            (* RETRY DISABLED - No retry count limit checking
            // Check if try count exceeds limit after incrementing
            // RetryCount specifies maximum number of attempts allowed
            // RetryCount=0 means 1 attempt, RetryCount=1 means 1 attempt, RetryCount=2 means 2 attempts, etc.
            IF (CommandStatus.CommandTryCount > _ResolveCommandConfiguration().RetryCount) AND
               (_ResolveCommandConfiguration().RetryCount > 0) THEN
                CommandStatus.Result := E_CommandResult.TooManyRequests; // 429
                // Log the TooManyRequests error with command details
                TraceWithSeverity(
                    Message := Tc2_Standard.CONCAT('Command exceeded retry limit: ',
                        Tc2_Standard.CONCAT(CommandStatus.LastCommandMessage,
                        Tc2_Standard.CONCAT(' | TryCount: ',
                        Tc2_Standard.CONCAT(DINT_TO_STRING(CommandStatus.CommandTryCount),
                        Tc2_Standard.CONCAT(' | RetryLimit: ',
                        DINT_TO_STRING(_ResolveCommandConfiguration().RetryCount)))))),
                    Severity := Global.TcEventSeverity.Warning);
                IF __ISVALIDREF(CommandStatus.BaseStatus) THEN
                    CommandStatus.BaseStatus.Error := TRUE;
                                        CommandStatus.BaseStatus.Done := TRUE;  // Complete state always sets Done=TRUE (terminal state)
                                    ELSE
                    TraceWithSeverity(Message := 'Command Base Reference Data Structure not present - see _InitializeReferences', Severity := Global.TcEventSeverity.Error);
                END_IF
                CommandStatus.StepState := E_CommandState.Complete;
                                //iTimer.ResetTimer();
            ELSIF (CommandStatus.CommandTryCount > 1) AND
                  (_ResolveCommandConfiguration().RetryCount = 0) THEN
                // Special case: RetryCount=0 means only 1 attempt allowed
                CommandStatus.Result := E_CommandResult.TooManyRequests; // 429
                // Log the TooManyRequests error for no-retry configuration
                TraceWithSeverity(
                    Message := Tc2_Standard.CONCAT('Command exceeded limit (no retries allowed): ',
                        Tc2_Standard.CONCAT(CommandStatus.LastCommandMessage,
                        Tc2_Standard.CONCAT(' | TryCount: ',
                        DINT_TO_STRING(CommandStatus.CommandTryCount)))),
                    Severity := Global.TcEventSeverity.Warning);
                IF __ISVALIDREF(CommandStatus.BaseStatus) THEN
                    CommandStatus.BaseStatus.Error := TRUE;
                                        CommandStatus.BaseStatus.Done := TRUE;  // Complete state always sets Done=TRUE (terminal state)
                                    ELSE
                    TraceWithSeverity(Message := 'Command Base Reference Data Structure not present - see _InitializeReferences', Severity := Global.TcEventSeverity.Error);
                END_IF
                CommandStatus.StepState := E_CommandState.Complete;
                                //iTimer.ResetTimer();
            END_IF
            *)
        END_IF

    E_CommandState.Execute:
        // Execute state: immediately transition to Monitor (tests expect this progression)
        CommandStatus.StepState := E_CommandState.Monitor;
        
    E_CommandState.Monitor:
        // All commands now monitor for completion condition
        // Check for timeout first (error condition takes priority)
        IF (_iCommandConfiguration <> 0) THEN
            IF CommandStatus.LastCommandElapsedTime >= TIME_TO_LTIME(_iCommandConfiguration.P_CommandConfiguration.TimeoutTime) THEN
                IF __ISVALIDREF(_iCommandConfiguration.P_CommandConfiguration.BaseConfiguration) THEN
                    IF _iCommandConfiguration.P_CommandConfiguration.BaseConfiguration.LogTraceConfiguration.What.xLogToEventLogger THEN
                        TraceWithSeverity(Message := 'Command timeout exceeded', Severity := Global.TcEventSeverity.Error);
                    END_IF
                END_IF
                Complete();  // Handle cleanup and clear Busy flag
                CommandStatus.Result := E_CommandResult.RequestTimeout;  // Override with timeout result
                                IF __ISVALIDREF(CommandStatus.BaseStatus) THEN
                    CommandStatus.BaseStatus.Error := TRUE;  // Set error flag for timeout
                                        CommandStatus.BaseStatus.Done := TRUE;  // Complete state always sets Done=TRUE (terminal state)
                                    ELSE
                    TraceWithSeverity(Message := 'Command Base Reference Data Structure not present - see _InitializeReferences', Severity := Global.TcEventSeverity.Error);
                END_IF
                CommandStatus.StepState := E_CommandState.Complete;  // Transition to Complete state
                            // Check if completion condition is met using resolved configuration (supports fallback)
            ELSIF __ISVALIDREF(_ResolveCommandConfiguration().CompletionCondition) AND_THEN
                  _ResolveCommandConfiguration().CompletionCondition THEN
                // Completion condition met - call Complete() to handle cleanup and transition
                IF NOT SUPER^.BaseStatus.LogTraceStatus.CompletionConditionMetShown THEN
                    TraceWithSeverity(Message := 'Completion condition met', Severity := Global.TcEventSeverity.Info);
                    SUPER^.BaseStatus.LogTraceStatus.CompletionConditionMetShown := TRUE;
                END_IF
                Complete();
                // Set Done flag and Ok result for successful completion (since Complete state won't be processed in this cycle due to REPEAT..UNTIL)
                IF CommandStatus.Result = E_CommandResult.Accepted THEN
                    CommandStatus.Result := E_CommandResult.Ok;
                    IF __ISVALIDREF(CommandStatus.BaseStatus) THEN
                        CommandStatus.BaseStatus.Done := TRUE;
                    ELSE
                        TraceWithSeverity(Message := 'Command Base Reference Data Structure not present - see _InitializeReferences', Severity := Global.TcEventSeverity.Error);
                    END_IF
                END_IF
                CommandStatus.StepState := E_CommandState.Complete;
                            END_IF
        ELSE
            // WARNING: _iCommandConfiguration is null - timeout monitoring disabled, relying on completion condition only
            TraceWithSeverity(Message := 'WARNING: _iCommandConfiguration is null in Monitor state - timeout monitoring disabled', Severity := Global.TcEventSeverity.Warning);
            IF __ISVALIDREF(_ResolveCommandConfiguration().CompletionCondition) AND_THEN
               _ResolveCommandConfiguration().CompletionCondition THEN
			   IF NOT SUPER^.BaseStatus.LogTraceStatus.CompletionConditionMetShown THEN
			       TraceWithSeverity(Message := 'Completion condition met', Severity := Global.TcEventSeverity.Info);
			       SUPER^.BaseStatus.LogTraceStatus.CompletionConditionMetShown := TRUE;
			   END_IF
                // No command configuration but completion condition met
                Complete();
                // Set Done flag and Ok result for successful completion (since Complete state won't be processed in this cycle due to REPEAT..UNTIL)
                IF CommandStatus.Result = E_CommandResult.Accepted THEN
                    CommandStatus.Result := E_CommandResult.Ok;
                    IF __ISVALIDREF(CommandStatus.BaseStatus) THEN
                        CommandStatus.BaseStatus.Done := TRUE;
                    ELSE
                        TraceWithSeverity(Message := 'Command Base Reference Data Structure not present - see _InitializeReferences', Severity := Global.TcEventSeverity.Error);
                    END_IF
                END_IF
                CommandStatus.StepState := E_CommandState.Complete;
                            END_IF
        END_IF
        // Otherwise stay in Monitor state until:
        // 1. CompletionCondition becomes TRUE
        // 2. Component calls Complete() method directly
        // 3. Timeout occurs (checked above)

    E_CommandState.Complete:
        // Stop the timer when entering Complete state
        IF iTimer <> 0 THEN
            iTimer.StopTimer();
        END_IF

        // Only set Ok on successful completion (if no error was already set)
        IF CommandStatus.Result = E_CommandResult.Accepted THEN
            CommandStatus.Result := E_CommandResult.Ok;
                        IF __ISVALIDREF(CommandStatus.BaseStatus) THEN
                CommandStatus.BaseStatus.Done := TRUE;
                            ELSE
                TraceWithSeverity(Message := 'Command Base Reference Data Structure not present - see _InitializeReferences', Severity := Global.TcEventSeverity.Error);
            END_IF
        END_IF
        // Otherwise preserve the existing error result (RequestTimeout, Aborted, etc.)
        // Error results already have Done=TRUE set by the method that created the error


END_CASE
UNTIL (CommandStatus.StepState = E_CommandState.Monitor) OR
      (CommandStatus.StepState = E_CommandState.Complete) OR
      (CommandStatus.StepState = E_CommandState.Idle)
END_REPEAT
END_METHOD

METHOD PRIVATE _ResetCommand
// Policy G: Always clear to complete reset state
IF __ISVALIDREF(CommandStatus.BaseStatus) THEN
	// Verbose logging: Log reset with context before clearing state
	TraceWithSeverity(
		Message := CONCAT(
			CONCAT('Resetting command from StepState: ', _FormatStepStateString(CommandStatus.StepState)),
			CONCAT(' | Result: ', CONCAT(_FormatResultString(CommandStatus.Result),
			CONCAT(' | TryCount: ', DINT_TO_STRING(CommandStatus.CommandTryCount))))
		),
		Severity := Global.TcEventSeverity.Verbose
	);

	CommandStatus.CommandTryCount	:= 0;
	CommandStatus.BaseStatus.Busy	:= FALSE;
	CommandStatus.Result 			:= E_CommandResult.None;
	CommandStatus.BaseStatus.Done	:= FALSE;
	CommandStatus.BaseStatus.Error	:= FALSE;
	CommandStatus.BaseStatus.ErrorID := 0; // Clear error ID per policy G
	CommandStatus.StepState			:= E_CommandState.Idle;
	CommandStatus.PreviousStepState := E_CommandState.Idle; // Reset previous state tracking

	// Reset Complete state cycle counter
	CompleteStateCycles := 0;

	// Reset the command timer to clear elapsed time
	IF iTimer <> 0 THEN
		iTimer.ResetTimer();
	ELSE
		// Timer interface not available - log critical error
		TraceWithSeverity(Message := 'CRITICAL: Timer interface not available during _ResetCommand - elapsed time may not reset!', Severity := Global.TcEventSeverity.Error);
	END_IF

	// Force reset elapsed time tracking to prevent instant timeout on next execution
	// This is a backup in case iTimer is null and ResetTimer() couldn't clear these
	CommandStatus.LastCommandElapsedTime := LTIME#0s;
	CommandStatus.LastCommandTriggerTime := 0;

	// Reset cyclic log spam flags to allow messages on next execution
	CommandStatus.BaseStatus.LogTraceStatus.CmdValidatedShown := FALSE;
	CommandStatus.BaseStatus.LogTraceStatus.CmdValidationFailedShown := FALSE;
	CommandStatus.BaseStatus.LogTraceStatus.CompletionConditionMetShown := FALSE;
	CommandStatus.BaseStatus.LogTraceStatus.InterlockLossShown := FALSE;
	CommandStatus.BaseStatus.LogTraceStatus.ConfigInvalidRefShown := FALSE;
ELSE
	TraceWithSeverity(Message := 'Command Base Reference Data Structure not present - see _InitializeReferences', Severity := Global.TcEventSeverity.Error);
END_IF
END_METHOD

METHOD PROTECTED _ResolveCommandConfiguration : REFERENCE TO ST_CommandConfiguration
VAR
    logEnabled : BOOL;
END_VAR
// Precompute whether we should emit logs
logEnabled := (SUPER^.BaseConfiguration.LogTraceConfiguration.When = E_LogTraceWhen.xRunCyclic)
              AND_THEN SUPER^.BaseConfiguration.LogTraceConfiguration.What.xLogToEventLogger;

// 1) Missing command interface?
IF _iCommandConfiguration = 0 THEN
    IF SUPER^.BaseConfiguration.LogTraceConfiguration.What.xLogToEventLogger AND NOT SUPER^.BaseStatus.LogTraceStatus.ConfigInvalidRefShown THEN
        TraceWithSeverity('Missing I_CommandConfiguration interface', Severity := Global.TcEventSeverity.Error);
        SUPER^.BaseStatus.LogTraceStatus.ConfigInvalidRefShown := TRUE;
    END_IF

// 2) Missing perm-intlk interface?
ELSIF _iPermIntlkConfiguration = 0 THEN
    IF SUPER^.BaseConfiguration.LogTraceConfiguration.What.xLogToEventLogger AND NOT SUPER^.BaseStatus.LogTraceStatus.ConfigInvalidRefShown THEN
        TraceWithSeverity('Missing I_PermIntlkConfiguration interface', Severity := Global.TcEventSeverity.Error);
        SUPER^.BaseStatus.LogTraceStatus.ConfigInvalidRefShown := TRUE;
    END_IF

ELSE
    // Both interfaces non-zero → validate each link in the chain

    // a) Command POU config must exist
    IF NOT __ISVALIDREF(_iCommandConfiguration.P_CommandConfiguration) THEN
        IF SUPER^.BaseConfiguration.LogTraceConfiguration.What.xLogToEventLogger AND NOT SUPER^.BaseStatus.LogTraceStatus.ConfigInvalidRefShown THEN
            TraceWithSeverity('_iCommandConfiguration.P_CommandConfiguration is invalid', Severity := Global.TcEventSeverity.Error);
            SUPER^.BaseStatus.LogTraceStatus.ConfigInvalidRefShown := TRUE;
        END_IF

    // b) PermIntlk POU config must exist
    ELSIF NOT __ISVALIDREF(_iPermIntlkConfiguration.P_PermIntlkConfiguration) THEN
        IF __ISVALIDREF(_iCommandConfiguration.P_CommandConfiguration.BaseConfiguration) THEN
            IF _iCommandConfiguration.P_CommandConfiguration.BaseConfiguration.LogTraceConfiguration.What.xLogToEventLogger AND NOT SUPER^.BaseStatus.LogTraceStatus.ConfigInvalidRefShown THEN
                TraceWithSeverity('_iPermIntlkConfiguration.P_PermIntlkConfiguration is invalid', Severity := Global.TcEventSeverity.Error);
                SUPER^.BaseStatus.LogTraceStatus.ConfigInvalidRefShown := TRUE;
            END_IF
        ELSE
            IF SUPER^.BaseConfiguration.LogTraceConfiguration.What.xLogToEventLogger AND NOT SUPER^.BaseStatus.LogTraceStatus.ConfigInvalidRefShown THEN
                TraceWithSeverity('_iPermIntlkConfiguration.P_PermIntlkConfiguration is invalid', Severity := Global.TcEventSeverity.Error);
                SUPER^.BaseStatus.LogTraceStatus.ConfigInvalidRefShown := TRUE;
            END_IF
        END_IF

    // c) Command BaseConfiguration must exist
    ELSIF NOT __ISVALIDREF(_iCommandConfiguration.P_CommandConfiguration.BaseConfiguration) THEN
        IF SUPER^.BaseConfiguration.LogTraceConfiguration.What.xLogToEventLogger AND NOT SUPER^.BaseStatus.LogTraceStatus.ConfigInvalidRefShown THEN
            TraceWithSeverity('_iCommandConfiguration.P_CommandConfiguration.BaseConfiguration is invalid', Severity := Global.TcEventSeverity.Warning);
            SUPER^.BaseStatus.LogTraceStatus.ConfigInvalidRefShown := TRUE;
        END_IF

    // d) PermIntlk BaseConfiguration must exist
    ELSIF NOT __ISVALIDREF(_iPermIntlkConfiguration.P_PermIntlkConfiguration.BaseConfiguration) THEN
        IF __ISVALIDREF(_iCommandConfiguration.P_CommandConfiguration.BaseConfiguration) THEN
            IF _iCommandConfiguration.P_CommandConfiguration.BaseConfiguration.LogTraceConfiguration.What.xLogToEventLogger AND NOT SUPER^.BaseStatus.LogTraceStatus.ConfigInvalidRefShown THEN
                TraceWithSeverity('_iPermIntlkConfiguration.P_PermIntlkConfiguration.BaseConfiguration is invalid', Severity := Global.TcEventSeverity.Error);
                SUPER^.BaseStatus.LogTraceStatus.ConfigInvalidRefShown := TRUE;
            END_IF
        ELSE
            IF SUPER^.BaseConfiguration.LogTraceConfiguration.What.xLogToEventLogger AND NOT SUPER^.BaseStatus.LogTraceStatus.ConfigInvalidRefShown THEN
                TraceWithSeverity('_iPermIntlkConfiguration.P_PermIntlkConfiguration.BaseConfiguration is invalid', Severity := Global.TcEventSeverity.Error);
                SUPER^.BaseStatus.LogTraceStatus.ConfigInvalidRefShown := TRUE;
            END_IF
        END_IF

    // e) Command InstancePath must exist
    ELSIF NOT __ISVALIDREF(_iCommandConfiguration.P_CommandConfiguration.BaseConfiguration.InstancePath) THEN
        IF __ISVALIDREF(_iCommandConfiguration.P_CommandConfiguration.BaseConfiguration) THEN
            IF _iCommandConfiguration.P_CommandConfiguration.BaseConfiguration.LogTraceConfiguration.What.xLogToEventLogger AND NOT SUPER^.BaseStatus.LogTraceStatus.ConfigInvalidRefShown THEN
                TraceWithSeverity('_iCommandConfiguration.P_CommandConfiguration.BaseConfiguration.InstancePath is invalid', Severity := Global.TcEventSeverity.Error);
                SUPER^.BaseStatus.LogTraceStatus.ConfigInvalidRefShown := TRUE;
            END_IF
        ELSE
            IF SUPER^.BaseConfiguration.LogTraceConfiguration.What.xLogToEventLogger AND NOT SUPER^.BaseStatus.LogTraceStatus.ConfigInvalidRefShown THEN
                TraceWithSeverity('_iCommandConfiguration.P_CommandConfiguration.BaseConfiguration.InstancePath is invalid', Severity := Global.TcEventSeverity.Error);
                SUPER^.BaseStatus.LogTraceStatus.ConfigInvalidRefShown := TRUE;
            END_IF
        END_IF

    // f) PermIntlk InstancePath must exist
    ELSIF NOT __ISVALIDREF(_iPermIntlkConfiguration.P_PermIntlkConfiguration.BaseConfiguration.InstancePath) THEN
        IF __ISVALIDREF(_iCommandConfiguration.P_CommandConfiguration.BaseConfiguration) THEN
            IF _iCommandConfiguration.P_CommandConfiguration.BaseConfiguration.LogTraceConfiguration.What.xLogToEventLogger AND NOT SUPER^.BaseStatus.LogTraceStatus.ConfigInvalidRefShown THEN
                TraceWithSeverity('_iPermIntlkConfiguration.P_PermIntlkConfiguration.BaseConfiguration.InstancePath is invalid', Severity := Global.TcEventSeverity.Error);
                SUPER^.BaseStatus.LogTraceStatus.ConfigInvalidRefShown := TRUE;
            END_IF
        ELSE
            IF SUPER^.BaseConfiguration.LogTraceConfiguration.What.xLogToEventLogger AND NOT SUPER^.BaseStatus.LogTraceStatus.ConfigInvalidRefShown THEN
                TraceWithSeverity('_iPermIntlkConfiguration.P_PermIntlkConfiguration.BaseConfiguration.InstancePath is invalid', Severity := Global.TcEventSeverity.Error);
                SUPER^.BaseStatus.LogTraceStatus.ConfigInvalidRefShown := TRUE;
            END_IF
        END_IF

    ELSE
        // All injected refs are valid — wire them up and return
        _iCommandConfiguration.P_CommandConfiguration.PermIntlkConfiguration 
          REF= _iPermIntlkConfiguration.P_PermIntlkConfiguration;
        _ResolveCommandConfiguration
          REF= _iCommandConfiguration.P_CommandConfiguration;
        CommandStatus.CmdConfigurationResolution   := E_ConfigurationResolution.InjectedInterface;
        CommandStatus.PermIntlkConfigResolution   := E_ConfigurationResolution.InjectedInterface;
        RETURN;
    END_IF

END_IF

// Fallback when any check failed
_ResolveCommandConfiguration REF= LocalCommandConfiguration;
CommandStatus.CmdConfigurationResolution   := E_ConfigurationResolution.Local;
CommandStatus.PermIntlkConfigResolution   := E_ConfigurationResolution.Local;
IF SUPER^.BaseConfiguration.LogTraceConfiguration.What.xLogToEventLogger THEN
    TraceWithSeverity('Using fallback CommandConfiguration', Severity := Global.TcEventSeverity.Info);
END_IF
END_METHOD

METHOD PRIVATE _ResolveCommandStatus : REFERENCE TO ST_CommandStatus
IF CommandStatus.CmdConfigurationResolution = E_ConfigurationResolution.InjectedInterface THEN
	IF _iCommandConfiguration <> 0 THEN
		CommandStatus.ConfigRef REF= _iCommandConfiguration.P_CommandConfiguration;
	END_IF
ELSE
	//Fallback
	CommandStatus.ConfigRef REF= LocalCommandConfiguration;
	IF SUPER^.BaseConfiguration.LogTraceConfiguration.When = E_LogTraceWhen.xRunCyclic AND_THEN 
		SUPER^.BaseConfiguration.LogTraceConfiguration.What.xLogToEventLogger THEN
			TraceWithSeverity(Message := 'Using fallback CommandConfiguration', Severity := Global.TcEventSeverity.Info);
	END_IF
END_IF

_ResolveCommandStatus REF= CommandStatus;
END_METHOD

METHOD PRIVATE _ResolvePermIntlkConfiguration : REFERENCE TO ST_PermIntlkConfiguration
VAR
    logEnabled : BOOL;
END_VAR
// 0) Precompute “should we log?”
logEnabled := (SUPER^.BaseConfiguration.LogTraceConfiguration.When = E_LogTraceWhen.xRunCyclic)
              AND_THEN SUPER^.BaseConfiguration.LogTraceConfiguration.What.xLogToEventLogger;

// 1) No injected interface?
IF _iPermIntlkConfiguration = 0 THEN
    IF SUPER^.BaseConfiguration.LogTraceConfiguration.What.xLogToEventLogger THEN
        TraceWithSeverity('Missing I_PermIntlkConfiguration interface', Severity := Global.TcEventSeverity.Error);
    END_IF

ELSE
    // Only now that _iPermIntlkConfiguration<>0 do we inspect its fields:

    // 2) Does the injected P_PermIntlkConfiguration pointer itself exist?
    IF NOT __ISVALIDREF(_iPermIntlkConfiguration.P_PermIntlkConfiguration) THEN
        IF SUPER^.BaseConfiguration.LogTraceConfiguration.What.xLogToEventLogger THEN
            TraceWithSeverity('_iPermIntlkConfiguration.P_PermIntlkConfiguration is invalid', Severity := Global.TcEventSeverity.Info);
        END_IF

    // 3) Is its BaseConfiguration valid?
    ELSIF NOT __ISVALIDREF(_iPermIntlkConfiguration.P_PermIntlkConfiguration.BaseConfiguration) THEN
        IF SUPER^.BaseConfiguration.LogTraceConfiguration.What.xLogToEventLogger THEN
            TraceWithSeverity('_iPermIntlkConfiguration.P_PermIntlkConfiguration.BaseConfiguration is invalid', Severity := Global.TcEventSeverity.Info);
        END_IF

    // 4) Is its BaseConfiguration.InstancePath valid?
    ELSIF NOT __ISVALIDREF(_iPermIntlkConfiguration.P_PermIntlkConfiguration.BaseConfiguration.InstancePath) THEN
        IF SUPER^.BaseConfiguration.LogTraceConfiguration.What.xLogToEventLogger THEN
            TraceWithSeverity('_iPermIntlkConfiguration.P_PermIntlkConfiguration.BaseConfiguration.InstancePath is invalid', Severity := Global.TcEventSeverity.Info);
        END_IF

    ELSE
        // 5) All injected refs are valid → use it and return
        _ResolvePermIntlkConfiguration 
          REF= _iPermIntlkConfiguration.P_PermIntlkConfiguration;
        CommandStatus.PermIntlkConfigResolution := E_ConfigurationResolution.InjectedInterface;
        RETURN;
    END_IF
END_IF

// 6) Fallback: use local config
_ResolvePermIntlkConfiguration REF= LocalPermIntlkConfiguration;
CommandStatus.PermIntlkConfigResolution    := E_ConfigurationResolution.Local;
IF SUPER^.BaseConfiguration.LogTraceConfiguration.What.xLogToEventLogger THEN
    TraceWithSeverity('Using fallback PermIntlkConfiguration', Severity := Global.TcEventSeverity.Info);
END_IF
END_METHOD

METHOD PROTECTED _UpdateComponentStatus
// Update component with last command executed (if component is available)
IF _iComponent <> 0 THEN
	IF CommandStatus.LastCommandResult <> CommandStatus.Result THEN
		CommandStatus.LastCommandResult := CommandStatus.Result;
		_iComponent.P_ComponentStatus.iLastCommand := THIS^;
	END_IF
ELSE
	// Warning: Component interface not available - cannot update component status
	TraceWithSeverity(Message := 'Warning: _iComponent is null in _UpdateComponentStatus - component status not updated', Severity := Global.TcEventSeverity.Warning);
END_IF
END_METHOD

METHOD PROTECTED _UpdateStatusEdgeTracking
// Override base class method to add CommandStatus-specific edge detection
// This method performs edge detection for both BaseStatus (via SUPER^) and CommandStatus
// Call parent class implementation for BaseStatus edge detection
SUPER^._UpdateStatusEdgeTracking();

// Only perform CommandStatus edge detection if verbose tracing is enabled
IF GPL_Base.PERSISTENT_LOG_LEVEL_MIN > Global.TcEventSeverity.Verbose THEN
	RETURN; // Skip edge detection if verbose level is not enabled
END_IF

// StepState edge detection
IF CommandStatus.StepState <> PreviousCommandStatus.StepState THEN
	TraceWithSeverity(
		Message := CONCAT(
			CONCAT('CommandStatus.StepState: ', _FormatStepStateString(PreviousCommandStatus.StepState)),
			CONCAT(' -> ', _FormatStepStateString(CommandStatus.StepState))
		),
		Severity := Global.TcEventSeverity.Verbose
	);
	PreviousCommandStatus.StepState := CommandStatus.StepState;
END_IF

// Result edge detection
IF CommandStatus.Result <> PreviousCommandStatus.Result THEN
	TraceWithSeverity(
		Message := CONCAT(
			CONCAT('CommandStatus.Result: ', _FormatResultString(PreviousCommandStatus.Result)),
			CONCAT(' -> ', _FormatResultString(CommandStatus.Result))
		),
		Severity := Global.TcEventSeverity.Verbose
	);
	PreviousCommandStatus.Result := CommandStatus.Result;
END_IF

// LastCommandTriggerTime edge detection (command start or reset)
IF CommandStatus.LastCommandTriggerTime <> PreviousCommandStatus.LastCommandTriggerTime THEN
	IF CommandStatus.LastCommandTriggerTime = 0 THEN
		// Trigger time reset to 0 - command has been reset
		TraceWithSeverity(
			Message := 'Command Reset - LastCommandTriggerTime cleared',
			Severity := Global.TcEventSeverity.Verbose
		);
	ELSE
		// Trigger time set to actual time - command has started
		TraceWithSeverity(
			Message := CONCAT(
				'Command Started - LastCommandTriggerTime: ',
				F_FileTimeToString(CommandStatus.LastCommandTriggerTime)
			),
			Severity := Global.TcEventSeverity.Verbose
		);
	END_IF
	PreviousCommandStatus.LastCommandTriggerTime := CommandStatus.LastCommandTriggerTime;
END_IF

// LastCommandCompletionTime edge detection (command complete)
IF CommandStatus.LastCommandCompletionTime <> PreviousCommandStatus.LastCommandCompletionTime THEN
	TraceWithSeverity(
		Message := CONCAT(
			CONCAT('Command Completed - LastCommandCompletionTime: ',
			F_FileTimeToString(CommandStatus.LastCommandCompletionTime)),
			CONCAT(' | ElapsedTime: ', LTIME_TO_STRING(CommandStatus.LastCommandElapsedTime))
		),
		Severity := Global.TcEventSeverity.Verbose
	);
	PreviousCommandStatus.LastCommandCompletionTime := CommandStatus.LastCommandCompletionTime;
END_IF
END_METHOD

METHOD PRIVATE _ValidateCommand
VAR
    maxRetries    : DINT;
    isBusy        : BOOL;
    hasPermissive : BOOL := TRUE;
    traceMessage  : STRING;
END_VAR
// Resolve configuration parameters - uses fallback if injected config is invalid
// RETRY DISABLED: maxRetries := _ResolveCommandConfiguration().RetryCount;

// Check component busy state
isBusy := (_iComponent <> 0) AND_THEN _iComponent.Busy;

// Check component enabled state - disabled components cannot execute commands
IF (_iComponent <> 0) AND_THEN NOT _iComponent.P_BaseStatus.Enabled THEN
    CommandStatus.Result := E_CommandResult.Forbidden;    // 403
        IF __ISVALIDREF(CommandStatus.BaseStatus) THEN
        CommandStatus.BaseStatus.Error := TRUE;
            ELSE
        TraceWithSeverity(Message := 'Command Base Reference Data Structure not present - see _InitializeReferences', Severity := Global.TcEventSeverity.Error);
    END_IF
    traceMessage := 'Component disabled - command execution forbidden';
    RETURN;
END_IF

// Check permissives based on configuration availability
// Allow fallback to local configuration when injected config is missing
IF (_iPermIntlkConfiguration <> 0) AND_THEN
   __ISVALIDREF(_iPermIntlkConfiguration.P_PermIntlkConfiguration) AND
   (iPermIntlk <> 0) THEN
    // Injected permissive configuration available
    IF iPermIntlk.Initialized THEN
        // Ensure permissive is current - CyclicLogic now handles evaluation automatically
        iPermIntlk.CyclicLogic();
        hasPermissive := iPermIntlk.P_OK;
        traceMessage := 'Permissive evaluated based on injected configuration';
    ELSE
        // Allow execution if permissive interface provided but not initialized (fail-open for basic tests)
        hasPermissive := TRUE;
        traceMessage := 'Permissive interface present but not initialized - allowing execution';
    END_IF
ELSE
    // No injected permissive config - use fallback (allow execution)
    hasPermissive := TRUE;
    traceMessage := 'Using local fallback configuration – allowing execution';
END_IF

// Now perform validation checks in order of priority
(* RETRY DISABLED - No retry count validation
// Only check retry count if this is actually a retry (command not in Idle state)
IF (CommandStatus.StepState <> E_CommandState.Idle) AND (CommandStatus.CommandTryCount > maxRetries) THEN
    CommandStatus.Result := E_CommandResult.TooManyRequests; // 429
    // Log the validation failure for too many requests
    TraceWithSeverity(
        Message := Tc2_Standard.CONCAT('Command validation failed - retry count exceeded: ',
            Tc2_Standard.CONCAT(CommandStatus.LastCommandMessage,
            Tc2_Standard.CONCAT(' | TryCount: ',
            Tc2_Standard.CONCAT(DINT_TO_STRING(CommandStatus.CommandTryCount),
            Tc2_Standard.CONCAT(' | MaxRetries: ',
            DINT_TO_STRING(maxRetries)))))),
        Severity := Global.TcEventSeverity.Warning);
    IF __ISVALIDREF(CommandStatus.BaseStatus) THEN
        CommandStatus.BaseStatus.Error := TRUE;  // Set error flag for too many requests
            ELSE
        TraceWithSeverity(Message := 'Command Base Reference Data Structure not present - see _InitializeReferences', Severity := Global.TcEventSeverity.Error);
    END_IF
    traceMessage := 'Retry count exceeded';
ELSIF *)
IF (CommandStatus.StepState = E_CommandState.Idle) AND isBusy THEN
    // Only check component busy when starting from Idle (prevents conflicts with other commands)
    // When resuming from Paused/etc, component will be busy with THIS command, which is expected
    CommandStatus.Result := E_CommandResult.BadRequest;        // 400
        IF __ISVALIDREF(CommandStatus.BaseStatus) THEN
        CommandStatus.BaseStatus.Error := TRUE;  // Set error flag for bad request
            ELSE
        TraceWithSeverity(Message := 'Command Base Reference Data Structure not present - see _InitializeReferences', Severity := Global.TcEventSeverity.Error);
    END_IF
    traceMessage := 'Component busy';
ELSIF NOT hasPermissive THEN
    CommandStatus.Result := E_CommandResult.Forbidden;       // 403
    	IF __ISVALIDREF(CommandStatus.BaseStatus) THEN
  		CommandStatus.BaseStatus.Error := TRUE;  // Set error flag for forbidden
  	ELSE
		TraceWithSeverity(Message := 'Command Base Reference Data Structure not present - see _InitializeReferences', Severity := Global.TcEventSeverity.Error);
	END_IF
    IF traceMessage = '' THEN
        traceMessage := 'Permissive not satisfied';
    END_IF
ELSE
    // Policy H: Do NOT increment try count here - only on actual execution start
    CommandStatus.Result := E_CommandResult.Accepted;      // 202
        IF __ISVALIDREF(CommandStatus.BaseStatus) THEN
        CommandStatus.BaseStatus.Error := FALSE;  // Clear error flag for successful validation
            ELSE
        TraceWithSeverity(Message := 'Command Base Reference Data Structure not present - see _InitializeReferences', Severity := Global.TcEventSeverity.Error);
    END_IF
    traceMessage := 'Validation succeeded – ready to process/queue';
END_IF

// Trace logging if enabled
IF _iCommandConfiguration <> 0 THEN
	IF __ISVALIDREF(_iCommandConfiguration.P_CommandConfiguration.BaseConfiguration) THEN
		IF _iCommandConfiguration.P_CommandConfiguration.BaseConfiguration.LogTraceConfiguration.When = E_LogTraceWhen.xRunCyclic AND_THEN
		   _iCommandConfiguration.P_CommandConfiguration.BaseConfiguration.LogTraceConfiguration.What.xLogToEventLogger THEN

			// Only log validation failures once to prevent spam
			IF (CommandStatus.Result <> E_CommandResult.Accepted) THEN
				IF NOT SUPER^.BaseStatus.LogTraceStatus.CmdValidationFailedShown THEN
					TraceWithSeverity(Message :=
						Tc2_Standard.CONCAT(
							STR1 := TO_STRING(CommandStatus.Result),
							STR2 := Tc2_Standard.CONCAT(STR1 := '; ', STR2 := traceMessage)
						), Severity := Global.TcEventSeverity.Info
					);
					SUPER^.BaseStatus.LogTraceStatus.CmdValidationFailedShown := TRUE;
				END_IF
			ELSE
				// Log successful validation normally (less spam concern)
				TraceWithSeverity(Message :=
					Tc2_Standard.CONCAT(
						STR1 := TO_STRING(CommandStatus.Result),
						STR2 := Tc2_Standard.CONCAT(STR1 := '; ', STR2 := traceMessage)
					), Severity := Global.TcEventSeverity.Info
				);
			END_IF
		END_IF
	ELSE
		TraceWithSeverity(Message := 'P_CommandConfiguration.BaseConfiguration reference invalid in _ValidateCommand method', Severity := Global.TcEventSeverity.Error);
		RETURN;
	END_IF
ELSE
	// WARNING: Validation trace logging disabled - configuration interface is null
	TraceWithSeverity(Message := 'WARNING: _iCommandConfiguration is null in _ValidateCommand - validation trace logging disabled', Severity := Global.TcEventSeverity.Warning);
END_IF
END_METHOD

METHOD CyclicLogic
SUPER^.CyclicLogic();

fbPermIntlk.CyclicLogic();

// Only update timer if interface is available
IF iTimer <> 0 THEN
	fbCmdElapsedTime.CyclicLogic();
ELSE
	// Log error once if timer interface is missing during active command
	IF (CommandStatus.StepState <> E_CommandState.Idle) AND (CommandStatus.StepState <> E_CommandState.Complete) THEN
		TraceWithSeverity(Message := 'CRITICAL: Timer interface not present during active command execution!', Severity := Global.TcEventSeverity.Error);
	END_IF
END_IF

// Track state changes for other purposes (CommandTryCount persists across retries, only cleared by Reset)
IF CommandStatus.PreviousStepState <> CommandStatus.StepState THEN
    CommandStatus.PreviousStepState := CommandStatus.StepState;
END_IF

// Execute state machine progression
_ProcessStateTransitions();

// Update component with last command result
_UpdateComponentStatus();

// Handle auto-reset for successful completions
_HandleAutoReset();

// Monitor interlocks and timeouts
_MonitorInterlocks();

// Perform edge detection for status changes at end of cycle (includes BaseStatus and CommandStatus)
_UpdateStatusEdgeTracking();
END_METHOD

PROPERTY P_CommandConfiguration : REFERENCE TO ST_CommandConfiguration
GET
P_CommandConfiguration REF= _ResolveCommandConfiguration();
END_GET
END_PROPERTY

PROPERTY P_PermIntlkConfiguration : REFERENCE TO ST_PermIntlkConfiguration
GET
P_PermIntlkConfiguration REF= _ResolvePermIntlkConfiguration();
END_GET
END_PROPERTY

END_FUNCTION_BLOCK

// PermIntlk/POUs/FB_PermIntlkCommand
{attribute 'no_explicit_call' := 'do not call this POU directly'}
{attribute 'enable_dynamic_creation'}
FUNCTION_BLOCK FB_PermIntlkCommand EXTENDS FB_PermIntlk
VAR
 	_iCommandConfiguration		: I_CommandConfiguration; // External Dependency
END_VAR

METHOD CyclicLogic
SUPER^.CyclicLogic();
END_METHOD

METHOD InjectCommandConfiguration
VAR_INPUT
    iCommandCfg 	: REFERENCE TO I_CommandConfiguration;
END_VAR
IF iCommandCfg = 0 THEN
	//Can't access Trace configuration on Init; use base config
		IF BaseConfiguration.LogTraceConfiguration.What.xLogToEventLogger THEN
			TraceWithSeverity(Message := 'Null Injected interface for Command Configuration!', Severity := Global.TcEventSeverity.Error);
		END_IF
    RETURN;
END_IF

_iCommandConfiguration := iCommandCfg;
END_METHOD

END_FUNCTION_BLOCK

// PermIntlk/POUs/FB_PermIntlk
{attribute 'no_explicit_call' := 'do not call this POU directly'}
{attribute 'enable_dynamic_creation'}
FUNCTION_BLOCK FB_PermIntlk EXTENDS FB_BaseCyclic IMPLEMENTS I_PermIntlk, I_PermIntlkConfiguration
VAR
 	_iPermIntlkConfiguration	: I_PermIntlkConfiguration; // External Dependency
	PermIntlkConfiguration 		: ST_PermIntlkConfiguration; //Local Reference Fallback	
	PermIntlkIndex				: DINT; // FOR loop, etc.
	PermIntlkLogIndex			: DINT; // FOR loop, etc.
	PermIntlkStatus 			: ST_PermIntlkStatus;

	// Guard flag to prevent duplicate evaluation in same scan
	evaluatedThisScan			: BOOL := FALSE;

	// Dummy interface instances for __QUERYINTERFACE type checking
	iQueryInterfaceCheckPermIntlkConfiguration	: I_PermIntlkConfiguration;
END_VAR

METHOD Evaluate : I_PermIntlk
CyclicLogic();

Evaluate := THIS^;
END_METHOD

{attribute 'monitoring' := 'call'}
PROPERTY FINAL P_OK : BOOL
GET
// Ensure fresh evaluation before returning status (avoid duplicate calls in same scan)
IF NOT evaluatedThisScan THEN
    _EvaluateOK();
    evaluatedThisScan := TRUE;
END_IF
P_OK := _ResolvePermIntlkStatus().PermIntlkOK;
END_GET
END_PROPERTY

PROPERTY P_PermIntlkConfiguration : REFERENCE TO ST_PermIntlkConfiguration
GET
P_PermIntlkConfiguration REF= _ResolvePermIntlkConfiguration();
END_GET
END_PROPERTY

(* Basic component initialization logic*)
METHOD PROTECTED _Initialize : BOOL
VAR
	InterimInit : BOOL;
END_VAR
// Initialize children dependencies first
InterimInit := _InitializeChildrenDependencies();
IF NOT InterimInit THEN
	IF PermIntlkConfiguration.BaseConfiguration.LogTraceConfiguration.What.xLogToEventLogger AND NOT PermIntlkStatus.BaseStatus.LogTraceStatus.InitChildrenFailureShown THEN
		TraceWithSeverity(Message := Tc2_Standard.CONCAT('_InitializeChildrenDependencies Failed at ', __POUNAME()), Severity := Global.TcEventSeverity.Error);
		PermIntlkStatus.BaseStatus.LogTraceStatus.InitChildrenFailureShown := TRUE;
	END_IF
	_Initialize := FALSE;
	RETURN;
END_IF

// Set element indices and resolve configurations
_SetElementIndices();
_ResolvePermIntlkConfiguration();
_ResolvePermIntlkStatus();

// Initialize references second
InterimInit := _InitializeReferences();
IF NOT InterimInit THEN
	IF PermIntlkConfiguration.BaseConfiguration.LogTraceConfiguration.What.xLogToEventLogger AND NOT PermIntlkStatus.BaseStatus.LogTraceStatus.InitReferencesFailureShown THEN
		TraceWithSeverity(Message := Tc2_Standard.CONCAT('_InitializeReferences Failed at ', __POUNAME()), Severity := Global.TcEventSeverity.Error);
		PermIntlkStatus.BaseStatus.LogTraceStatus.InitReferencesFailureShown := TRUE;
	END_IF
	_Initialize := FALSE;
	RETURN;
END_IF

// Set dependency configuration last
InterimInit := _SetDependencyConfiguration();
IF NOT InterimInit THEN
	IF PermIntlkConfiguration.BaseConfiguration.LogTraceConfiguration.What.xLogToEventLogger AND NOT PermIntlkStatus.BaseStatus.LogTraceStatus.InitDependencyConfigFailureShown THEN
		TraceWithSeverity(Message := Tc2_Standard.CONCAT('_SetDependencyConfiguration Failed at ', __POUNAME()), Severity := Global.TcEventSeverity.Error);
		PermIntlkStatus.BaseStatus.LogTraceStatus.InitDependencyConfigFailureShown := TRUE;
	END_IF
	_Initialize := FALSE;
	RETURN;
END_IF

// All initialization steps succeeded
_Initialize := TRUE;
END_METHOD

METHOD PROTECTED _InitializeReferences : BOOL
//Order is important!
BaseConfiguration.InstancePath 					REF= InstancePath;

PermIntlkConfiguration.BaseConfiguration		REF= SUPER^.BaseConfiguration;

PermIntlkStatus.BaseStatus						REF= SUPER^.BaseStatus;

// Use resolved configuration for setting up references
IF PermIntlkStatus.PermIntlkConfigResolution = E_ConfigurationResolution.InjectedInterface THEN
	IF _iPermIntlkConfiguration <> 0 THEN
		PermIntlkConfiguration := _iPermIntlkConfiguration.P_PermIntlkConfiguration;
	END_IF
	PermIntlkStatus.ConfigRef	REF= _iPermIntlkConfiguration.P_PermIntlkConfiguration.PermIntlkObj;
	FOR PermIntlkIndex := GC_PermIntlk.INDEX_CONDITION_MIN TO GC_PermIntlk.INDEX_CONDITION_MAX BY 1 DO
		PermIntlkStatus.ConditionStatus[PermIntlkIndex].PermObj	REF= _iPermIntlkConfiguration.P_PermIntlkConfiguration.PermIntlkObj[PermIntlkIndex];
	END_FOR
ELSE
	PermIntlkStatus.ConfigRef	REF= PermIntlkConfiguration.PermIntlkObj;
	FOR PermIntlkIndex := GC_PermIntlk.INDEX_CONDITION_MIN TO GC_PermIntlk.INDEX_CONDITION_MAX BY 1 DO
		PermIntlkConfiguration.PermIntlkObj[PermIntlkIndex].Condition REF= PermIntlkStatus.PermIntlkConditionAlwaysFalse;
		PermIntlkStatus.ConditionStatus[PermIntlkIndex].PermObj	REF= PermIntlkConfiguration.PermIntlkObj[PermIntlkIndex];
	END_FOR
END_IF

_InitializeReferences 							:= TRUE; // apply at end of all reference initialization
END_METHOD

METHOD PROTECTED _SetElementIndices
IF (_iPermIntlkConfiguration <> 0) AND __QUERYINTERFACE(_iPermIntlkConfiguration, iQueryInterfaceCheckPermIntlkConfiguration) THEN
	FOR PermIntlkIndex := GC_PermIntlk.INDEX_CONDITION_MIN TO GC_PermIntlk.INDEX_CONDITION_MAX BY 1 DO
		IF _iPermIntlkConfiguration.P_PermIntlkConfiguration.PermIntlkObj[PermIntlkIndex].Index = 0 THEN
			_iPermIntlkConfiguration.P_PermIntlkConfiguration.PermIntlkObj[PermIntlkIndex].Index := PermIntlkIndex;
		END_IF
	END_FOR
END_IF
END_METHOD

METHOD PRIVATE _EvaluateConfiguration
VAR
	resolvedConfig : REFERENCE TO ST_PermIntlkConfiguration;
	previousResolution : E_ConfigurationResolution;
END_VAR
// Store previous resolution to detect changes
previousResolution := PermIntlkStatus.PermIntlkConfigResolution;

// Get the resolved configuration (injected or local)
resolvedConfig REF= _ResolvePermIntlkConfiguration();

// If configuration resolution changed, update references
IF PermIntlkStatus.PermIntlkConfigResolution <> previousResolution THEN
	_InitializeReferences();
END_IF

FOR PermIntlkLogIndex := GC_PermIntlk.INDEX_CONDITION_MIN TO GC_PermIntlk.INDEX_CONDITION_MAX BY 1 DO

	IF (resolvedConfig.PermIntlkObj[PermIntlkLogIndex].Description <> '') AND
		(resolvedConfig.PermIntlkObj[PermIntlkLogIndex].Description <> 'PermIntlk Condition Not Configured') THEN
		PermIntlkStatus.ConditionStatus[PermIntlkLogIndex].Configured := TRUE;
	END_IF

	//Evaluate Permissive Condition=>Status - references already set up in _InitializeReferences
	_LogMessage(Index := PermIntlkLogIndex);

END_FOR
END_METHOD

METHOD PRIVATE _EvaluateOK
VAR_INST
	PermOKMsgTrig		: Tc2_Standard.R_TRIG;
	PermIntlkLostTrig	: Tc2_Standard.F_TRIG;
END_VAR
VAR
	hasConfiguredConditions : BOOL := FALSE;
	resolvedConfig : REFERENCE TO ST_PermIntlkConfiguration;
END_VAR
// Get the resolved configuration (injected or local)
resolvedConfig REF= _ResolvePermIntlkConfiguration();

// Initialize result based on mode
IF resolvedConfig.Mode = E_ModePermIntlk.IfAnyConditionMet THEN
	PermIntlkStatus.PermIntlkOK := FALSE; // In "Any" mode, assume FALSE until we find a TRUE condition
ELSE
	PermIntlkStatus.PermIntlkOK := TRUE;  // In "All" mode, assume TRUE until we find a FALSE condition
END_IF

FOR PermIntlkIndex := GC_PermIntlk.INDEX_CONDITION_MIN TO GC_PermIntlk.INDEX_CONDITION_MAX BY 1 DO
	
	IF __ISVALIDREF(PermIntlkStatus.ConditionStatus[PermIntlkIndex].PermObj) AND PermIntlkStatus.ConditionStatus[PermIntlkIndex].Configured THEN
		
		IF __ISVALIDREF(PermIntlkStatus.ConditionStatus[PermIntlkIndex].PermObj.Condition) THEN
			hasConfiguredConditions := TRUE;
			IF resolvedConfig.Mode = E_ModePermIntlk.IfAllConditionsMet THEN
				IF NOT PermIntlkStatus.ConditionStatus[PermIntlkIndex].PermObj.Condition THEN
					PermIntlkStatus.PermIntlkOK := FALSE;				
					EXIT;
				END_IF
			ELSIF resolvedConfig.Mode = E_ModePermIntlk.IfAnyConditionMet THEN
				IF PermIntlkStatus.ConditionStatus[PermIntlkIndex].PermObj.Condition THEN
					PermIntlkStatus.PermIntlkOK := TRUE;				
					EXIT;
				END_IF
			END_IF
		ELSE
			PermIntlkStatus.ConditionStatus[PermIntlkIndex].PermObj.Condition REF= PermIntlkStatus.PermIntlkConditionAlwaysFalse;
			TraceWithSeverity(Message := 'Using Injected Interface, but no valid condition reference was supplied - PermIntlk Default Failure', Severity := Global.TcEventSeverity.Error);
		END_IF
	END_IF

END_FOR

// If no configured conditions exist, default to TRUE (safe state)
IF NOT hasConfiguredConditions THEN
	PermIntlkStatus.PermIntlkOK := TRUE;
END_IF

IF SUPER^.BaseConfiguration.LogTraceConfiguration.When = E_LogTraceWhen.xRunCyclic AND_THEN
	SUPER^.BaseConfiguration.LogTraceConfiguration.What.xLogToEventLogger THEN

		PermOKMsgTrig(CLK := PermIntlkStatus.PermIntlkOK);
		PermIntlkLostTrig(CLK := NOT PermIntlkStatus.PermIntlkOK);

		IF PermOKMsgTrig.Q THEN
			SUPER^.TraceWithSeverity(Message := 'Permissive OK ', Severity := Global.TcEventSeverity.Info);
		END_IF

		IF PermIntlkLostTrig.Q THEN
			SUPER^.TraceWithSeverity(Message := 'Interlock Lost ', Severity := Global.TcEventSeverity.Error);
		END_IF

END_IF
END_METHOD

METHOD PROTECTED _LogMessage
VAR_INPUT
	Index : DINT;
END_VAR
//Build output message
IF SUPER^.BaseConfiguration.LogTraceConfiguration.When = E_LogTraceWhen.xRunCyclic AND_THEN
		SUPER^.BaseConfiguration.LogTraceConfiguration.What.xLogToEventLogger THEN
			IF __ISVALIDREF(PermIntlkStatus.ConditionStatus[Index].PermObj) THEN
				// Check if Condition reference is valid before accessing it
				IF __ISVALIDREF(PermIntlkStatus.ConditionStatus[Index].PermObj.Condition) THEN
					IF NOT PermIntlkStatus.ConditionStatus[Index].PermObj.Condition THEN
						IF PermIntlkStatus.ConditionStatus[Index].Configured THEN
							IF NOT PermIntlkStatus.BaseStatus.LogTraceStatus.PermIntlkConditionFailureShown THEN
								PermIntlkStatus.ConditionStatus[Index].ConditionMessage := 'Permissive Condition Missing: ';
								_PermMsgIndexForMessage(Index := Index);
								PermIntlkStatus.ConditionStatus[Index].ConditionMessage := Tc2_Standard.CONCAT(STR1 := PermIntlkStatus.ConditionStatus[Index].ConditionMessage, STR2 := ' ');
								PermIntlkStatus.ConditionStatus[Index].ConditionMessage := Tc2_Standard.CONCAT(STR1 := PermIntlkStatus.ConditionStatus[Index].ConditionMessage, STR2 := PermIntlkStatus.ConditionStatus[Index].PermObj.Description);
								SUPER^.TraceWithSeverity(Message := PermIntlkStatus.ConditionStatus[Index].ConditionMessage, Severity := Global.TcEventSeverity.Error);
								PermIntlkStatus.BaseStatus.LogTraceStatus.PermIntlkConditionFailureShown := TRUE;
							END_IF
						ELSE
							IF NOT PermIntlkStatus.BaseStatus.LogTraceStatus.PermIntlkConditionFailureShown THEN
								PermIntlkStatus.ConditionStatus[Index].ConditionMessage := 'Permissive Description Missing.  Configure permissive: ';
								_PermMsgIndexForMessage(Index := Index);
								SUPER^.TraceWithSeverity(Message := PermIntlkStatus.ConditionStatus[Index].ConditionMessage, Severity := Global.TcEventSeverity.Warning);
								PermIntlkStatus.BaseStatus.LogTraceStatus.PermIntlkConditionFailureShown := TRUE;
							END_IF
						END_IF
					END_IF
				ELSE
					// Condition reference is invalid
					IF PermIntlkStatus.ConditionStatus[Index].Configured THEN
						IF NOT PermIntlkStatus.BaseStatus.LogTraceStatus.PermIntlkConditionFailureShown THEN
							PermIntlkStatus.ConditionStatus[Index].ConditionMessage := 'Permissive Condition Reference Invalid for Index: ';
							_PermMsgIndexForMessage(Index := Index);
							SUPER^.TraceWithSeverity(Message := PermIntlkStatus.ConditionStatus[Index].ConditionMessage, Severity := Global.TcEventSeverity.Error);
							PermIntlkStatus.BaseStatus.LogTraceStatus.PermIntlkConditionFailureShown := TRUE;
						END_IF
					END_IF
				END_IF
			END_IF
// ELSE // logs a message regardless of configuration, due to critical Permissive Data Reference missing
// 	PermIntlkStatus.PermissiveStatusMessage := 'Permissive Missing Reference to Component Log Trace Configuration.  Initialize Component Permissive Data Reference';
// 	SUPER^.Trace(Message := PermIntlkStatus.PermissiveStatusMessage);
END_IF
END_METHOD

METHOD PROTECTED _PermMsgIndexForMessage
VAR_INPUT
	Index : DINT;
END_VAR
PermIntlkStatus.ConditionStatus[Index].ConditionMessage := Tc2_Standard.CONCAT(STR1 := PermIntlkStatus.ConditionStatus[Index].ConditionMessage, STR2 := ' Index:');				
PermIntlkStatus.ConditionStatus[Index].ConditionMessage := Tc2_Standard.CONCAT(STR1 := PermIntlkStatus.ConditionStatus[Index].ConditionMessage, STR2 := UDINT_TO_STRING(PermIntlkStatus.ConditionStatus[Index].PermObj.Index));
END_METHOD

METHOD PROTECTED _ResolvePermIntlkConfiguration : REFERENCE TO ST_PermIntlkConfiguration
VAR
    logEnabled : BOOL;
END_VAR
// Precompute whether we should log
logEnabled := (SUPER^.BaseConfiguration.LogTraceConfiguration.When = E_LogTraceWhen.xRunCyclic)
              AND_THEN SUPER^.BaseConfiguration.LogTraceConfiguration.What.xLogToEventLogger;

// If no interface at all, log and fall through to fallback
IF _iPermIntlkConfiguration = 0 THEN
    IF logEnabled THEN
        TraceWithSeverity('Missing I_PermIntlkConfiguration interface', Severity := Global.TcEventSeverity.Error);
    END_IF

ELSE
    // Only now that _iPermIntlkConfiguration<>0 do we inspect its fields:
    IF NOT __ISVALIDREF(_iPermIntlkConfiguration.P_PermIntlkConfiguration) THEN
        IF logEnabled THEN
            TraceWithSeverity('_iPermIntlkConfiguration.P_PermIntlkConfiguration is invalid', Severity := Global.TcEventSeverity.Info);
        END_IF

    // Optional: BaseConfiguration validation (non-blocking for basic functionality)
    ELSIF NOT __ISVALIDREF(_iPermIntlkConfiguration.P_PermIntlkConfiguration.BaseConfiguration) THEN
        IF logEnabled THEN
            TraceWithSeverity('BaseConfiguration is invalid - using injected interface anyway', Severity := Global.TcEventSeverity.Warning);
        END_IF
        // Continue to use injected interface despite missing BaseConfiguration
        _ResolvePermIntlkConfiguration REF= _iPermIntlkConfiguration.P_PermIntlkConfiguration;
        PermIntlkStatus.PermIntlkConfigResolution := E_ConfigurationResolution.InjectedInterface;
        RETURN;

    ELSIF NOT __ISVALIDREF(_iPermIntlkConfiguration.P_PermIntlkConfiguration.BaseConfiguration.InstancePath) THEN
        IF logEnabled THEN
            TraceWithSeverity('InstancePath is invalid - using injected interface anyway', Severity := Global.TcEventSeverity.Warning);
        END_IF
        // Continue to use injected interface despite missing InstancePath
        _ResolvePermIntlkConfiguration REF= _iPermIntlkConfiguration.P_PermIntlkConfiguration;
        PermIntlkStatus.PermIntlkConfigResolution := E_ConfigurationResolution.InjectedInterface;
        RETURN;

    ELSE
        // All injected refs are valid → return it
        _ResolvePermIntlkConfiguration REF= _iPermIntlkConfiguration.P_PermIntlkConfiguration;
        PermIntlkStatus.PermIntlkConfigResolution := E_ConfigurationResolution.InjectedInterface;
        RETURN;
    END_IF
END_IF

// Fallback path when either interface=0 or any validity check failed:
_ResolvePermIntlkConfiguration REF= PermIntlkConfiguration;
PermIntlkStatus.PermIntlkConfigResolution := E_ConfigurationResolution.Local;
IF logEnabled THEN
    TraceWithSeverity('Using fallback PermIntlkConfiguration', Severity := Global.TcEventSeverity.Info);
END_IF
END_METHOD

METHOD PROTECTED _ResolvePermIntlkStatus : REFERENCE TO ST_PermIntlkStatus
// FOR PermIntlkIndex := LOWER_BOUND(PermIntlkStatus.ConditionStatus,1) TO UPPER_BOUND(PermIntlkStatus.ConditionStatus,1) BY 1 DO
// 	IF __ISVALIDREF(PermIntlkStatus.BaseStatus) AND __ISVALIDREF(PermIntlkStatus.ConfigRef) AND __ISVALIDREF(PermIntlkStatus.ConditionStatus[PermIntlkIndex].PermObj) THEN
// 		_ResolvePermIntlkStatus REF= PermIntlkStatus;		
// 	END_IF
// END_FOR

IF PermIntlkStatus.PermIntlkConfigResolution = E_ConfigurationResolution.InjectedInterface THEN
	PermIntlkStatus.ConfigRef REF= _iPermIntlkConfiguration.P_PermIntlkConfiguration.PermIntlkObj;
ELSE
	PermIntlkStatus.ConfigRef REF= PermIntlkConfiguration.PermIntlkObj;
END_IF

_ResolvePermIntlkStatus REF= PermIntlkStatus;
END_METHOD

METHOD PROTECTED _ConfigurationCyclic
SUPER^._ConfigurationCyclic();

_EvaluateConfiguration();
END_METHOD

METHOD CyclicLogic
SUPER^.CyclicLogic();

// Reset guard flag at start of new scan cycle
evaluatedThisScan := FALSE;

// Always evaluate permissive state on every cycle
_EvaluateOK();
evaluatedThisScan := TRUE;
END_METHOD

METHOD InjectPermIntlkConfiguration
VAR_INPUT
    iPermIntlkCfg 	: I_PermIntlkConfiguration;
END_VAR
// Allow injecting null to clear the interface (for runtime config loss scenarios)
_iPermIntlkConfiguration := iPermIntlkCfg;

IF iPermIntlkCfg = 0 THEN
	//Log warning about null interface - will fall back to local configuration
		TraceWithSeverity(Message := 'Null Injected interface for PermIntlk Configuration - using local fallback', Severity := Global.TcEventSeverity.Warning);
END_IF
END_METHOD

PROPERTY P_PermIntlkStatus : REFERENCE TO ST_PermIntlkStatus
GET
P_PermIntlkStatus REF= PermIntlkStatus;
END_GET
END_PROPERTY

METHOD ReinitObjects
VAR
	 InitPermIntlk 	: ST_PermIntlkConfigurationCondition;
END_VAR
FOR PermIntlkIndex := GC_PermIntlk.INDEX_CONDITION_MIN TO GC_PermIntlk.INDEX_CONDITION_MAX DO
	InitPermIntlk.Condition REF= PermIntlkStatus.PermIntlkConditionAlwaysFalse;
	PermIntlkConfiguration.PermIntlkObj[PermIntlkIndex]	:= InitPermIntlk;
END_FOR
PermIntlkStatus.PermIntlkOK := TRUE;

// Reset cyclic log spam flag to allow messages after reinit
PermIntlkStatus.BaseStatus.LogTraceStatus.PermIntlkConditionFailureShown := FALSE;
END_METHOD

END_FUNCTION_BLOCK

// Command/POUs/FB_CommandElapsedTimer
{attribute 'no_explicit_call' := 'do not call this POU directly'}
FUNCTION_BLOCK FB_CommandElapsedTimer EXTENDS FB_BaseCyclic IMPLEMENTS I_BaseCyclic, I_Timer //I_TestClock
VAR
	_iCommand					: I_Command; // External Dependency
	_iCommandConfiguration		: I_CommandConfiguration; // External Dependency
	sCfgLogMessage				: STRING := ' Timed Out';
	rtBusy 						: Tc2_Standard.R_TRIG;
	ftBusy 						: Tc2_Standard.F_TRIG;
	ftPaused					: Tc2_Standard.F_TRIG;
	Timer						: Tc2_Standard.TON := (PT := Tc2_System.Global_Variables.DEFAULT_ADS_TIMEOUT);
END_VAR

PROPERTY P_ElapsedTime : TIME
GET
P_ElapsedTime	:= Timer.ET;
END_GET
END_PROPERTY

PROPERTY P_IsElapsed : BOOL
GET
P_IsElapsed := (Timer.ET = Timer.PT);
END_GET
END_PROPERTY

METHOD ResetTimer
Timer.IN	:= FALSE;

// Clear elapsed time tracking to prevent stale values on next execution
IF _iCommand <> 0 THEN
	_iCommand.P_CommandStatus.LastCommandTriggerTime := 0;
	_iCommand.P_CommandStatus.LastCommandElapsedTime := LTIME#0s;
END_IF
END_METHOD

METHOD StartTimer
Timer.IN	:= TRUE;
END_METHOD

METHOD StopTimer
VAR_INPUT
END_VAR
// Stop timer and capture final elapsed time
// Guard: Only calculate if LastCommandTriggerTime has been initialized (> 0) to prevent huge elapsed time values
IF Timer.IN AND (_iCommand <> 0) AND (_iCommand.P_CommandStatus.LastCommandTriggerTime > 0) THEN
	_iCommand.P_CommandStatus.LastCommandCompletionTime := Tc2_System.F_GetSystemTime();
	_iCommand.P_CommandStatus.LastCommandElapsedTime := F_FILETIME64_TO_LTIME(FileTime64 :=
													_iCommand.P_CommandStatus.LastCommandCompletionTime - _iCommand.P_CommandStatus.LastCommandTriggerTime);
END_IF
Timer.IN := FALSE;
END_METHOD

METHOD CyclicLogic
SUPER^.CyclicLogic();

IF (_iCommand <> 0) AND (_iCommandConfiguration <> 0) THEN
	
	IF rtBusy.Q THEN
		Timer.IN 	:= TRUE;
		_iCommand.P_CommandStatus.LastCommandTriggerTime	:= Tc2_System.F_GetSystemTime();
	END_IF
	
	// Only update elapsed time if not already in Complete state
	// Guard: Only calculate if LastCommandTriggerTime has been initialized (> 0) to prevent huge elapsed time values
	IF (ftBusy.Q OR Timer.Q) AND (_iCommand.P_CommandStatus.StepState <> E_CommandState.Complete) AND (_iCommand.P_CommandStatus.LastCommandTriggerTime > 0) THEN
		_iCommand.P_CommandStatus.LastCommandCompletionTime	:= Tc2_System.F_GetSystemTime();
		_iCommand.P_CommandStatus.LastCommandElapsedTime 	:= F_FILETIME64_TO_LTIME(FileTime64 :=
																_iCommand.P_CommandStatus.LastCommandCompletionTime - _iCommand.P_CommandStatus.LastCommandTriggerTime);
	END_IF

	// Continuously update elapsed time while timer is running (but not in Complete state)
	// Guard: Only calculate if LastCommandTriggerTime has been initialized (> 0) to prevent huge elapsed time values
	IF Timer.IN AND (_iCommand.P_CommandStatus.StepState <> E_CommandState.Complete) AND (_iCommand.P_CommandStatus.LastCommandTriggerTime > 0) THEN
		_iCommand.P_CommandStatus.LastCommandElapsedTime := F_FILETIME64_TO_LTIME(FileTime64 :=
														Tc2_System.F_GetSystemTime() - _iCommand.P_CommandStatus.LastCommandTriggerTime);
	END_IF

	IF Timer.Q THEN
		IF SUPER^.BaseConfiguration.LogTraceConfiguration.When = E_LogTraceWhen.xRunCyclic AND_THEN
			SUPER^.BaseConfiguration.LogTraceConfiguration.What.xLogToEventLogger THEN
				_iCommand.P_CommandStatus.LastCommandMessage := Tc2_Standard.CONCAT(STR1 := 'Command ', STR2 := _iCommandConfiguration.P_CommandConfiguration.CommandDescription);
				_iCommand.P_CommandStatus.LastCommandMessage := Tc2_Standard.CONCAT(STR1 := _iCommand.P_CommandStatus.LastCommandMessage, STR2 := sCfgLogMessage);
				TraceWithSeverity(Message := _iCommand.P_CommandStatus.LastCommandMessage, Severity := Global.TcEventSeverity.Info);
		END_IF
		Timer.IN	:= FALSE;	
	END_IF

	ftPaused(CLK := (_iCommand.P_CommandStatus.StepState = E_CommandState.Paused));
	rtBusy(CLK := _iCommand.P_CommandStatus.BaseStatus.Busy OR ftPaused.Q);
	ftBusy(CLK := _iCommand.P_CommandStatus.BaseStatus.Busy OR _iCommand.P_CommandStatus.StepState = E_CommandState.Paused);
	
	SUPER^.BaseStatus.Busy 	:= Timer.IN;
	SUPER^.BaseStatus.Done	:= Timer.Q;
	Timer(PT := _iCommandConfiguration.P_CommandConfiguration.TimeoutTime);
END_IF
END_METHOD

METHOD InjectConfiguration
VAR_INPUT
    iCommand 		: I_Command;
    iCommandConfiguration 	: I_CommandConfiguration;
END_VAR
// Inject interfaces (moved from FB_Init)
IF iCommand <> 0 THEN
	THIS^._iCommand := iCommand;
END_IF

IF iCommandConfiguration <> 0 THEN
	_iCommandConfiguration := iCommandConfiguration;
END_IF
END_METHOD

END_FUNCTION_BLOCK

// Functions/Time/F_FILETIME64_TO_LTIME
FUNCTION F_FILETIME64_TO_LTIME : LTIME
VAR_INPUT
	FileTime64 : Tc2_Utilities.T_FILETIME64;
END_VAR

F_FILETIME64_TO_LTIME := TO_LTIME(FileTime64*100); // LTIME units = ns; FileTime64 units = 100ns

END_FUNCTION

// Functions/Time/F_FileTimeToString
FUNCTION F_FileTimeToString : Tc2_System.T_MaxString
VAR_INPUT
	fileTime : Tc2_Utilities.T_FILETIME64;
END_VAR
VAR
	timeAsDt : DT;
END_VAR

timeAsDt := Tc2_Utilities.FILETIME64_TO_DT(fileTime := fileTime);
F_FileTimeToString := DT_TO_STRING(timeAsDt);

END_FUNCTION

// Component/POUs/FB_Component
FUNCTION_BLOCK ABSTRACT FB_Component 
VAR_GENERIC CONSTANT
	MinIndexComponentCmd			: DINT := GC_Component.INDEX_COMMAND_MIN;
    MaxIndexComponentCmd			: DINT := GC_Component.INDEX_COMMAND_MAX;
END_VAR

EXTENDS FB_BaseCyclic IMPLEMENTS I_ComponentFull
VAR
	iComponentInternal							: I_ComponentFull := THIS^;

	ComponentConfiguration						: ST_ComponentConfiguration;
	ComponentStatus								: ST_ComponentStatus;
	
	CommandIndexCyclic							: DINT; // FOR Loop, etc.
	CommandIndexExit							: DINT; // FOR Loop w/ Exit
	CommandPermIntlkConfiguration				: ARRAY[MinIndexComponentCmd..MaxIndexComponentCmd] OF FB_CmdPermIntlkConfiguration;
	Commands 									: ARRAY[MinIndexComponentCmd..MaxIndexComponentCmd] OF FB_Command;
	iCommands									: ARRAY[MinIndexComponentCmd..MaxIndexComponentCmd] OF I_Command;
	iCommandConfigurations						: ARRAY[MinIndexComponentCmd..MaxIndexComponentCmd] OF I_CommandConfiguration;
	CommandCompletionConditions					: ARRAY[MinIndexComponentCmd..MaxIndexComponentCmd] OF BOOL;
	
	CommandBuffer								: FB_RingBufferICmd;
	iRingBufferICmd								: I_RingBufferICmd := CommandBuffer;
	SystimeICmd									: ST_SystimeICmd;

	_SystemPermIntlk							: I_PermIntlk; // External Dependency
	
	_ControlMode								: I_ControlMode; // External Dependency
	
    GetAmsNetId              					: Tc2_Utilities.FB_GetLocalAmsNetId := (tTimeout := Tc2_System.Global_Variables.DEFAULT_ADS_TIMEOUT);

	//Prevent Double Call per scan
	ProcessCommandQueueCalled					: BOOL;
	
//Hash Table
	fbHashDJB2_PouName							: FB_Hash_djb2;
	iHashDJB2_PouName							: I_HashFunction := fbHashDJB2_PouName;

	HashTablePouName							: FB_HashTable;
	iHashTablePouName							: I_HashTableBase := HashTablePouName;

	// Track which commands have shown configuration warnings to prevent cyclic logging
	CommandConfigWarningShown					: ARRAY[MinIndexComponentCmd..MaxIndexComponentCmd] OF BOOL;
	
	FirstCycScan		: BOOL;
END_VAR

METHOD DequeueCommand : BOOL
VAR_INPUT
	CmdIndex	: DINT;
END_VAR
DequeueCommand := _DequeueCommand(CmdIndex := CmdIndex);
END_METHOD

METHOD EnqueueCommand
VAR_INPUT
	CmdIndex	: DINT;
END_VAR
_EnqueueCommand(CmdIndex := CmdIndex);
END_METHOD

METHOD ExecuteCommand : I_ComponentFull
VAR_INPUT
	CmdIndex	: DINT;
END_VAR

(*
IF CmdIndex >= LOWER_BOUND(SUPER^.Commands,1) AND CmdIndex <= UPPER_BOUND(SUPER^.Commands,1) THEN
	SUPER^.ExecuteCommand(CmdIndex := CmdIndex);
	
	IF SUPER^.iCommands[CmdIndex].P_CommandStatus.Result = E_HttpStatusCode.Ok THEN
		ZaberStatus.ZaberMethodDispatch	:= CmdIndex;
	END_IF
	
	_ExecuteCommandByIndexOneShot();
ELSE
	Trace(Message := Tc2_Standard.CONCAT(STR1 := DINT_TO_STRING(CmdIndex), STR2 := ' not within array bounds'));
END_IF

ExecuteCommand := THIS^;
*)
// Check for index bounds first
IF (CmdIndex < LOWER_BOUND(Commands, 1)) OR (CmdIndex > UPPER_BOUND(Commands, 1)) THEN
    IF __ISVALIDREF(ComponentConfiguration.BaseConfiguration) THEN
        IF ComponentConfiguration.BaseConfiguration.LogTraceConfiguration.What.xLogToEventLogger THEN
            TraceWithSeverity(Message := 'Command Index Out of Bounds', Severity := Global.TcEventSeverity.Warning);
        END_IF
    END_IF
    RETURN;
END_IF

// Check for missing command interface
IF iCommands[CmdIndex] = 0 THEN
    IF __ISVALIDREF(ComponentConfiguration.BaseConfiguration) THEN
        IF ComponentConfiguration.BaseConfiguration.LogTraceConfiguration.What.xLogToEventLogger THEN
            TraceWithSeverity(Message := 'Missing Command Interface', Severity := Global.TcEventSeverity.Warning);
        END_IF
    END_IF
    RETURN;
END_IF

// CommandPermIntlkConfiguration always exists as concrete array - no need to check

// Check if ring buffer is available
IF iRingBufferICmd = 0 THEN
    IF __ISVALIDREF(ComponentConfiguration.BaseConfiguration) THEN
        IF ComponentConfiguration.BaseConfiguration.LogTraceConfiguration.What.xLogToEventLogger THEN
            TraceWithSeverity(Message := 'Missing Command Queue Interface', Severity := Global.TcEventSeverity.Error);
        END_IF
    END_IF
    RETURN;
END_IF

// Validate command before enqueuing
iCommands[CmdIndex].Validate();

// Handle validation result - check reference validity first
IF iCommands[CmdIndex] <> 0 AND __ISVALIDREF(iCommands[CmdIndex].P_CommandStatus) THEN
    CASE iCommands[CmdIndex].P_CommandStatus.Result OF
        E_CommandResult.Accepted:
            _EnqueueCommand(CmdIndex := CmdIndex);
            // Attempt immediate dequeue if possible
            _DequeueCommand(CmdIndex := CmdIndex);
        
        E_CommandResult.Forbidden,
        E_CommandResult.TooManyRequests:
            // Command rejected - trace the reason
            IF __ISVALIDREF(ComponentConfiguration.BaseConfiguration) THEN
                IF ComponentConfiguration.BaseConfiguration.LogTraceConfiguration.What.xLogToEventLogger THEN
                    TraceWithSeverity(Message := Tc2_Standard.CONCAT('Command validation failed: ', UDINT_TO_STRING(iCommands[CmdIndex].P_CommandStatus.Result)),
                                     Severity := Global.TcEventSeverity.Info);
                END_IF
            END_IF
        
        ELSE
            // Unexpected validation result
            IF __ISVALIDREF(ComponentConfiguration.BaseConfiguration) THEN
                IF ComponentConfiguration.BaseConfiguration.LogTraceConfiguration.What.xLogToEventLogger THEN
                    TraceWithSeverity(Message := Tc2_Standard.CONCAT('Unexpected command validation result: ', UDINT_TO_STRING(iCommands[CmdIndex].P_CommandStatus.Result)),
                                     Severity := Global.TcEventSeverity.Warning);
                END_IF
            END_IF
    END_CASE
ELSE
    IF __ISVALIDREF(ComponentConfiguration.BaseConfiguration) THEN
        IF ComponentConfiguration.BaseConfiguration.LogTraceConfiguration.What.xLogToEventLogger THEN
            TraceWithSeverity(Message := 'Invalid command status reference during ExecuteCommand', Severity := Global.TcEventSeverity.Error);
        END_IF
    END_IF
END_IF

ExecuteCommand := THIS^;
END_METHOD

METHOD GetIndexByPOUName : UINT
VAR_INPUT
	NameIn	: T_MaxString;
END_VAR
VAR
    HashResult : UINT;
END_VAR
// Default to 0 (invalid index) for failure cases
GetIndexByPOUName := 0;

IF iHashTablePouName = 0 THEN
    IF __ISVALIDREF(ComponentConfiguration.BaseConfiguration) THEN
        IF ComponentConfiguration.BaseConfiguration.LogTraceConfiguration.What.xLogToEventLogger THEN
            TraceWithSeverity(Message := 'Hash table interface is NULL in GetIndexByPOUName', Severity := Global.TcEventSeverity.Error);
        END_IF
    END_IF
    RETURN;
END_IF

HashResult := iHashTablePouName.GetIndex(NameIn := NameIn);

// Hash table returns UINT#65535 for "not found"
IF HashResult = UINT#65535 THEN
    IF __ISVALIDREF(ComponentConfiguration.BaseConfiguration) THEN
        IF ComponentConfiguration.BaseConfiguration.LogTraceConfiguration.What.xLogToEventLogger THEN
            TraceWithSeverity(Message := Tc2_Standard.CONCAT('Hash table lookup failed for POUName: ', NameIn), Severity := Global.TcEventSeverity.Warning);
        END_IF
    END_IF
    // Return 0 to indicate failure
    RETURN;
ELSE
    GetIndexByPOUName := HashResult;
END_IF
END_METHOD

{warning 'Add method implementation '}
METHOD HMICommunication
END_METHOD

METHOD InjectCommandQueue
VAR_INPUT
	iCommandQueue : I_RingBufferICmd;
END_VAR
IF iCommandQueue <> 0 THEN
    iRingBufferICmd := iCommandQueue;
ELSE
    IF __ISVALIDREF(ComponentConfiguration.BaseConfiguration) THEN
        IF ComponentConfiguration.BaseConfiguration.LogTraceConfiguration.What.xLogToEventLogger THEN
            TraceWithSeverity(Message := 'Null or invalid command queue interface injected!', Severity := Global.TcEventSeverity.Error);
        END_IF
    END_IF
END_IF
END_METHOD

PROPERTY P_CommandQueue : I_RingBufferICmd
GET
IF iRingBufferICmd <> 0 THEN 
	P_CommandQueue := iRingBufferICmd;
END_IF
END_GET
END_PROPERTY

PROPERTY P_ComponentConfiguration : REFERENCE TO ST_ComponentConfiguration
GET
P_ComponentConfiguration REF= ComponentConfiguration;
END_GET
END_PROPERTY

PROPERTY P_ComponentStatus : REFERENCE TO ST_ComponentStatus
GET
P_ComponentStatus	REF= ComponentStatus;
END_GET
END_PROPERTY

METHOD Reset : E_CommandResult
IF ComponentConfiguration.ResetResetsAllCommands THEN
	ResetAllCommands();
END_IF
END_METHOD

METHOD ResetAllCommands : E_CommandResult
// Reset all commands in the component
FOR CommandIndexCyclic := LOWER_BOUND(Commands,1) TO UPPER_BOUND(Commands,1) DO
	IF iCommands[CommandIndexCyclic] <> 0 THEN
		iCommands[CommandIndexCyclic].Reset();
	END_IF
END_FOR

ResetAllCommands := E_CommandResult.Ok;
END_METHOD

(*! @summary Basic component initialization logic*)
METHOD PROTECTED _Initialize : BOOL
VAR
	InterimInit : BOOL;
END_VAR
// Initialize children dependencies first
InterimInit := _InitializeChildrenDependencies();
IF NOT InterimInit THEN
	IF __ISVALIDREF(ComponentConfiguration.BaseConfiguration) THEN
		IF ComponentConfiguration.BaseConfiguration.LogTraceConfiguration.What.xLogToEventLogger AND NOT ComponentStatus.BaseStatus.LogTraceStatus.InitChildrenFailureShown THEN
			TraceWithSeverity(Message := Tc2_Standard.CONCAT('_InitializeChildrenDependencies Failed at ', __POUNAME()), Severity := Global.TcEventSeverity.Error);
			ComponentStatus.BaseStatus.LogTraceStatus.InitChildrenFailureShown := TRUE;
		END_IF
	END_IF
	_Initialize := FALSE;
	RETURN;
END_IF

// Initialize references second
InterimInit := _InitializeReferences();
IF NOT InterimInit THEN
	IF __ISVALIDREF(ComponentConfiguration.BaseConfiguration) THEN
		IF ComponentConfiguration.BaseConfiguration.LogTraceConfiguration.What.xLogToEventLogger AND NOT ComponentStatus.BaseStatus.LogTraceStatus.InitReferencesFailureShown THEN
			TraceWithSeverity(Message := Tc2_Standard.CONCAT('_InitializeReferences Failed at ', __POUNAME()), Severity := Global.TcEventSeverity.Error);
			ComponentStatus.BaseStatus.LogTraceStatus.InitReferencesFailureShown := TRUE;
		END_IF
	END_IF
	_Initialize := FALSE;
	RETURN;
END_IF

// Obtain AmsNetId if required
IF InterimInit THEN
	// Validate references before accessing properties
	IF NOT __ISVALIDREF(ComponentConfiguration.BaseConfiguration) THEN
		_Initialize := FALSE;
		RETURN;
	END_IF

	IF ComponentConfiguration.AmsNetIdRequired AND_THEN NOT ComponentStatus.AmsNetIdIsValid THEN
		REPEAT
			_ObtainAmsNetId();
		UNTIL ComponentStatus.AmsNetIdIsValid OR GetAmsNetId.bError
		END_REPEAT;

		IF GetAmsNetId.bError THEN
			IF ComponentConfiguration.BaseConfiguration.LogTraceConfiguration.What.xLogToEventLogger THEN
				TraceWithSeverity(Message := 'Error: Component failed to obtain AmsNetId', Severity := Global.TcEventSeverity.Error);
			END_IF
			_Initialize := FALSE;
			RETURN;
		END_IF
	END_IF
END_IF

ComponentStatus.BaseStatus.Busy := FALSE;

// Build hash tables
InterimInit := _BuildTables();
IF NOT InterimInit THEN
	IF __ISVALIDREF(ComponentConfiguration.BaseConfiguration) THEN
		IF ComponentConfiguration.BaseConfiguration.LogTraceConfiguration.What.xLogToEventLogger THEN
			TraceWithSeverity(Message := Tc2_Standard.CONCAT('_BuildTables Failed at ', __POUNAME()), Severity := Global.TcEventSeverity.Error);
		END_IF
	END_IF
	_Initialize := FALSE;
	RETURN;
END_IF

// Set command permission interlock configuration
InterimInit := _SetCommandPermIntlkConfiguration();
IF NOT InterimInit THEN
	IF __ISVALIDREF(ComponentConfiguration.BaseConfiguration) THEN
		IF ComponentConfiguration.BaseConfiguration.LogTraceConfiguration.What.xLogToEventLogger THEN
			TraceWithSeverity(Message := Tc2_Standard.CONCAT('_SetCommandPermIntlkConfiguration Failed at ', __POUNAME()), Severity := Global.TcEventSeverity.Error);
		END_IF
	END_IF
	_Initialize := FALSE;
	RETURN;
END_IF

// Set dependency configuration last
InterimInit := _SetDependencyConfiguration();
IF NOT InterimInit THEN
	IF __ISVALIDREF(ComponentConfiguration.BaseConfiguration) THEN
		IF ComponentConfiguration.BaseConfiguration.LogTraceConfiguration.What.xLogToEventLogger THEN
			TraceWithSeverity(Message := Tc2_Standard.CONCAT('_SetDependencyConfiguration Failed at ', __POUNAME()), Severity := Global.TcEventSeverity.Error);
		END_IF
	END_IF
	_Initialize := FALSE;
	RETURN;
END_IF

// All initialization steps succeeded
_Initialize := TRUE;
END_METHOD

METHOD PROTECTED _InitializeChildrenDependencies : BOOL
// Initialize concrete configurations and wire directly to Commands
FOR CommandIndexCyclic := LOWER_BOUND(Commands,1) TO UPPER_BOUND(Commands,1) BY 1 DO

	// Inject configurations directly - TwinCAT auto-converts to interfaces
	Commands[CommandIndexCyclic].InjectConfigurations(
		iComponent := THIS^,
		iCommandConfiguration := CommandPermIntlkConfiguration[CommandIndexCyclic],
		iPermIntlkConfiguration := CommandPermIntlkConfiguration[CommandIndexCyclic]);
		
	CommandPermIntlkConfiguration[CommandIndexCyclic].Initialize();
	Commands[CommandIndexCyclic].Initialize();
END_FOR

CommandBuffer.Initialize();

fbHashDJB2_PouName.Initialize();
HashTablePouName.Initialize();

HashTablePouName.InjectHashFunction(iHashFunction := iHashDJB2_PouName);

_InitializeChildrenDependencies := TRUE;
END_METHOD

METHOD PROTECTED _InitializeReferences : BOOL
//Initialize data references
//Order is important!
BaseConfiguration.InstancePath 						REF= InstancePath;

ComponentConfiguration.BaseConfiguration 			REF= SUPER^.BaseConfiguration;

ComponentStatus.BaseStatus							REF= SUPER^.BaseStatus;

// Create reference from ComponentStatus.AmsNetId to ComponentConfiguration.AmsNetId
// ComponentStatus.AmsNetId is a REFERENCE TO T_AmsNetID
// ComponentConfiguration.AmsNetId is a T_AmsNetID (direct member)
ComponentStatus.AmsNetId							REF= ComponentConfiguration.AmsNetId;

_InitializeReferences 								:= TRUE; // apply at end of all reference initialization
END_METHOD

METHOD PROTECTED _SetCommandIndices : BOOL
FOR CommandIndexCyclic := LOWER_BOUND(CommandPermIntlkConfiguration, 1) TO UPPER_BOUND(CommandPermIntlkConfiguration, 1) DO
	IF NOT ComponentStatus.CommandConfigurationInjected THEN
		IF CommandPermIntlkConfiguration[CommandIndexCyclic].P_CommandConfiguration.CommandIndex = 0 THEN
			CommandPermIntlkConfiguration[CommandIndexCyclic].P_CommandConfiguration.CommandIndex := CommandIndexCyclic; //default to ordinal if not provided by the interface
		END_IF
	END_IF
END_FOR

_SetCommandIndices := TRUE;
END_METHOD

METHOD PROTECTED _SetCommandPermIntlkConfiguration : BOOL
VAR_INPUT
END_VAR
_SetCommandPermIntlkConfiguration	:= _SetCommandIndices();;
END_METHOD

//FB_Init is always available implicitly and it is used primarily for initialization.
//The return value is not evaluated. For a specific influence, you can also declare the
//methods explicitly and provide additional code there with the standard initialization
//code. You can evaluate the return value.
METHOD FB_Init: BOOL
VAR_INPUT
    bInitRetains: BOOL; // TRUE: the retain variables are initialized (reset warm / reset cold)
    bInCopyCode: BOOL;  // TRUE: the instance will be copied to the copy code afterward (online change)   
END_VAR
//Interface wiring
FOR CommandIndexCyclic := LOWER_BOUND(Commands,1) TO UPPER_BOUND(Commands,1) BY 1 DO
	iCommands[CommandIndexCyclic] 					:= Commands[CommandIndexCyclic];
	iCommandConfigurations[CommandIndexCyclic]		:= CommandPermIntlkConfiguration[CommandIndexCyclic];
END_FOR

FB_Init := TRUE;
END_METHOD

METHOD InjectCommandConfiguration : BOOL
VAR_IN_OUT
	iCommandConfiguration			: ARRAY[*] OF I_CommandConfiguration; // External Dependency			
END_VAR
InjectCommandConfiguration := _InjectCommandConfiguration(iCommandConfiguration := iCommandConfiguration);
END_METHOD

METHOD InjectPermIntlkConfiguration : BOOL
VAR_IN_OUT
	iPermIntlkConfiguration			: ARRAY[*] OF I_PermIntlkConfiguration; // External Dependency			
END_VAR
InjectPermIntlkConfiguration	:= _InjectPermIntlkConfiguration(iPermIntlkConfiguration := iPermIntlkConfiguration);
END_METHOD

METHOD InjectSystemInterfaces
VAR_INPUT
	SystemPermIntlk				: I_PermIntlk;
	ControlMode					: I_ControlMode;
END_VAR
// Inject system-level interfaces (moved from FB_Init)
IF (SystemPermIntlk <> 0) THEN
	THIS^._SystemPermIntlk := SystemPermIntlk;
END_IF

IF (ControlMode <> 0) THEN
	THIS^._ControlMode := ControlMode;
END_IF
END_METHOD

METHOD PROTECTED _BuildTables : BOOL;
VAR
    InsertedCount : DINT := 0;
    POUName : T_MaxString;
END_VAR
FOR CommandIndexCyclic := LOWER_BOUND(Commands,1) TO UPPER_BOUND(Commands,1) BY 1 DO
	IF iHashTablePouName <> 0 THEN
        POUName := CommandPermIntlkConfiguration[CommandIndexCyclic].P_CommandConfiguration.CommandPOUName;
        
        IF POUName <> '' THEN
            iHashTablePouName.Insert(IdxIn := DINT_TO_UINT(CommandIndexCyclic), NameIn := POUName);
            InsertedCount := InsertedCount + 1;

            IF __ISVALIDREF(ComponentConfiguration.BaseConfiguration) THEN
                IF ComponentConfiguration.BaseConfiguration.LogTraceConfiguration.What.xLogToEventLogger THEN
                    TraceWithSeverity(Message := Tc2_Standard.CONCAT('Hash table insert: "',
                                     Tc2_Standard.CONCAT(POUName,
                                     Tc2_Standard.CONCAT('" -> Index ', DINT_TO_STRING(CommandIndexCyclic)))),
                                     Severity := Global.TcEventSeverity.Info);
                END_IF
            END_IF
        END_IF
	END_IF
END_FOR

IF __ISVALIDREF(ComponentConfiguration.BaseConfiguration) THEN
    IF ComponentConfiguration.BaseConfiguration.LogTraceConfiguration.What.xLogToEventLogger THEN
        TraceWithSeverity(Message := Tc2_Standard.CONCAT('Hash table built with ',
                         Tc2_Standard.CONCAT(DINT_TO_STRING(InsertedCount), ' entries')),
                         Severity := Global.TcEventSeverity.Info);
    END_IF
END_IF

_BuildTables := TRUE;
END_METHOD

METHOD PROTECTED _ClearTempCmdObj
SystimeICmd.iCmd := 0;
SystimeICmd.iCmdCfg	:= 0;
SystimeICmd.systimestamp := 0;
END_METHOD

METHOD PROTECTED _CommandsCyclic
VAR
	bHasCmdInterface		: BOOL;
	bHasCmdCfgInterface		: BOOL;
	bHasPermIntlkInterface 	: BOOL;

	sMessagePart1 : STRING;
	sMessage      : STRING;
END_VAR
// ── Per-command cyclic work ────────────────────────────────────────────
FOR CommandIndexCyclic := LOWER_BOUND(Commands, 1) TO UPPER_BOUND(Commands, 1) DO

    iCommands[CommandIndexCyclic] := Commands[CommandIndexCyclic];

    bHasCmdInterface       := (iCommands[CommandIndexCyclic] <> 0);
    bHasCmdCfgInterface    := TRUE;  // Always exists - concrete array
    bHasPermIntlkInterface := TRUE;  // Always exists - concrete array

    IF bHasCmdInterface AND bHasCmdCfgInterface AND bHasPermIntlkInterface THEN
        // Check if command configuration was actually provided (not just default/empty values)
        IF iCommandConfigurations[CommandIndexCyclic] <> 0 AND_THEN
           (iCommandConfigurations[CommandIndexCyclic].P_CommandConfiguration.CommandDescription <> '' OR
            iCommandConfigurations[CommandIndexCyclic].P_CommandConfiguration.CommandPOUName <> '') THEN
            // Run cyclic logic for all commands to enable auto-reset mechanism
            // Commands with Ok result need cycling to auto-reset from Complete state
            // Commands with error results may also need cycling for cleanup
            Commands[CommandIndexCyclic].CyclicLogic();
        ELSE
            // Command configuration not provided - log warning only once using edge detection
            IF NOT CommandConfigWarningShown[CommandIndexCyclic] THEN
                IF __ISVALIDREF(ComponentConfiguration.BaseConfiguration) THEN
                    IF ComponentConfiguration.BaseConfiguration.LogTraceConfiguration.What.xLogToEventLogger THEN
                        TraceWithSeverity(
                            Message := Tc2_Standard.CONCAT('Command[',
                                      Tc2_Standard.CONCAT(DINT_TO_STRING(CommandIndexCyclic),
                                      '] has no valid configuration. Cyclic logic NOT being called. Please provide command configuration for all indices or adjust array bounds.')),
                            Severity := Global.TcEventSeverity.Warning);
                        CommandConfigWarningShown[CommandIndexCyclic] := TRUE;
                    END_IF
                END_IF
            END_IF
        END_IF
    ELSE
        // ── Optional trace of missing interfaces ──
        IF __ISVALIDREF(ComponentConfiguration.BaseConfiguration) THEN
            IF ComponentConfiguration.BaseConfiguration.LogTraceConfiguration.When = E_LogTraceWhen.xRunCyclic AND_THEN
               ComponentConfiguration.BaseConfiguration.LogTraceConfiguration.What.xLogToEventLogger THEN

                // build "Command[n] missing: …" using only the two STRING vars
                sMessagePart1 := Tc2_Standard.CONCAT(
                                    STR1 := 'Command[',
                                    STR2 := DINT_TO_STRING(CommandIndexCyclic)
                                 );
                sMessage := Tc2_Standard.CONCAT(STR1 := sMessagePart1, STR2 := '] missing: ');

                IF NOT bHasCmdInterface       THEN sMessage := Tc2_Standard.CONCAT(STR1 := sMessage, STR2 := 'Cmd ');        END_IF
                IF NOT bHasCmdCfgInterface    THEN sMessage := Tc2_Standard.CONCAT(STR1 := sMessage, STR2 := 'Cfg ');        END_IF
                IF NOT bHasPermIntlkInterface THEN sMessage := Tc2_Standard.CONCAT(STR1 := sMessage, STR2 := 'PermIntlk ');  END_IF

                IF __ISVALIDREF(ComponentConfiguration.BaseConfiguration) THEN
                    IF ComponentConfiguration.BaseConfiguration.LogTraceConfiguration.What.xLogToEventLogger THEN
                        TraceWithSeverity(Message := sMessage, Severity := Global.TcEventSeverity.Info);
                    END_IF
                END_IF   // e.g. "Command[3] missing: Cmd Cfg "
            END_IF
        END_IF
    END_IF
END_FOR

// ── Busy flag now calculated after command completion in _UpdateBusyStatus() ──
// ── Finally run the queue processor ────────────────────────────────────
_ProcessCommandQueue();
ProcessCommandQueueCalled := FALSE;
END_METHOD

METHOD PROTECTED _ComponentCyclic : I_ComponentFull
FOR CommandIndexCyclic := LOWER_BOUND(Commands, 1) TO UPPER_BOUND(Commands, 1) DO
	// Inject configurations directly - TwinCAT auto-converts to interfaces
	Commands[CommandIndexCyclic].InjectConfigurations(
		iComponent := THIS^,
		iCommandConfiguration := CommandPermIntlkConfiguration[CommandIndexCyclic],
		iPermIntlkConfiguration := CommandPermIntlkConfiguration[CommandIndexCyclic]);
END_FOR

// Note: _EvaluateCompletionConditions(), _MonitorCommandCompletion(), and _UpdateComponentStatus()
// are now called directly from CyclicLogic() in the correct order

_ComponentCyclic := THIS^;
END_METHOD

METHOD PROTECTED _DequeueCommand : BOOL
VAR_INPUT
	CmdIndex	: DINT;
END_VAR
// Defensive checks first
IF (CmdIndex < LOWER_BOUND(Commands, 1)) OR (CmdIndex > UPPER_BOUND(Commands, 1)) THEN
    _DequeueCommand := FALSE;
    RETURN;
END_IF

IF (iCommands[CmdIndex] = 0) OR (iRingBufferICmd = 0) THEN
    _DequeueCommand := FALSE;
    RETURN;
END_IF

// Only dequeue if component is idle and command was successfully enqueued
IF iCommands[CmdIndex] <> 0 AND 
   __ISVALIDREF(iCommands[CmdIndex].P_CommandStatus) AND
   iCommands[CmdIndex].P_CommandStatus.Result = E_CommandResult.Accepted AND 
   NOT ComponentStatus.BaseStatus.Busy AND
   iRingBufferICmd.P_RingBufferStatus.ObjectCountInBufferPrim > 0 THEN
	_ProcessCommandQueue();
	_DequeueCommand := TRUE;
ELSE
	_DequeueCommand := FALSE;
END_IF
END_METHOD

METHOD PROTECTED _DispatchValid : BOOL;
VAR_INPUT
	cmdIndex : DINT;
END_VAR
// Validate command index is within bounds
_DispatchValid := (cmdIndex >= LOWER_BOUND(Commands, 1)) AND
                  (cmdIndex <= UPPER_BOUND(Commands, 1));
END_METHOD

METHOD PROTECTED _EnqueueCommand
VAR_INPUT
	CmdIndex	: DINT;
END_VAR
// Ensure the ring buffer exists
IF iRingBufferICmd = 0 THEN
	IF __ISVALIDREF(ComponentConfiguration.BaseConfiguration) THEN
		IF ComponentConfiguration.BaseConfiguration.LogTraceConfiguration.What.xLogToEventLogger THEN
			TraceWithSeverity(Message := 'No ring buffer configured for Commands', Severity := Global.TcEventSeverity.Error);
		END_IF
	END_IF
    RETURN;
END_IF

// Validate command interface before proceeding
IF iCommands[CmdIndex] = 0 THEN
	IF __ISVALIDREF(ComponentConfiguration.BaseConfiguration) THEN
		IF ComponentConfiguration.BaseConfiguration.LogTraceConfiguration.What.xLogToEventLogger THEN
			TraceWithSeverity(Message := 'Command interface is null at index', Severity := Global.TcEventSeverity.Error);
		END_IF
	END_IF
	RETURN;
END_IF

// Prepare command object
SystimeICmd.iCmd    := iCommands[CmdIndex];
SystimeICmd.iCmdCfg := CommandPermIntlkConfiguration[CmdIndex];

// Add to buffer
iRingBufferICmd.AddObject(RefObject := SystimeICmd);

// Check if add was successful
IF NOT iRingBufferICmd.P_ObjectWasAdded THEN
	IF __ISVALIDREF(ComponentConfiguration.BaseConfiguration) THEN
		IF ComponentConfiguration.BaseConfiguration.LogTraceConfiguration.What.xLogToEventLogger THEN
			TraceWithSeverity(Message := 'Failed to add command to queue - buffer may be full', Severity := Global.TcEventSeverity.Error);
		END_IF
	END_IF
	_ClearTempCmdObj();
	RETURN;
END_IF

_ClearTempCmdObj();

// Mark as queued successfully only if actually added - validate reference before accessing
IF iCommands[CmdIndex] <> 0 AND __ISVALIDREF(iCommands[CmdIndex].P_CommandStatus) THEN
	iCommands[CmdIndex].P_CommandStatus.Result := E_CommandResult.Accepted; // 202 Accepted
ELSE
	IF __ISVALIDREF(ComponentConfiguration.BaseConfiguration) THEN
		IF ComponentConfiguration.BaseConfiguration.LogTraceConfiguration.What.xLogToEventLogger THEN
			TraceWithSeverity(Message := 'Invalid command status reference at index', Severity := Global.TcEventSeverity.Error);
		END_IF
	END_IF
END_IF

// Clear the added flag to prepare for next add operation
iRingBufferICmd.ClearStatusFlagAdded();
END_METHOD

(*
Example Implementation:
// Set completion conditions - commands complete immediately after transitioning to acting state
// This prevents the component from staying busy and blocking other commands
SUPER^.CommandCompletionConditions[INDEX_COMMAND_ABORT]            		:= (SequencerStatus.CurrentState = E_PackMLState.Aborting);
SUPER^.CommandCompletionConditions[INDEX_COMMAND_CLEAR]            		:= (SequencerStatus.CurrentState = E_PackMLState.Clearing);
SUPER^.CommandCompletionConditions[INDEX_COMMAND_COMPLETE]         		:= (SequencerStatus.CurrentState = E_PackMLState.Completing);
SUPER^.CommandCompletionConditions[INDEX_COMMAND_HOLD]             		:= (SequencerStatus.CurrentState = E_PackMLState.Holding);
SUPER^.CommandCompletionConditions[INDEX_COMMAND_RESET]            		:= (SequencerStatus.CurrentState = E_PackMLState.Resetting);
SUPER^.CommandCompletionConditions[INDEX_COMMAND_RESUMEFROMHOLD]   		:= (SequencerStatus.CurrentState = E_PackMLState.Unholding);
SUPER^.CommandCompletionConditions[INDEX_COMMAND_RESUMEFROMSUSPEND]		:= (SequencerStatus.CurrentState = E_PackMLState.Unsuspending);
SUPER^.CommandCompletionConditions[INDEX_COMMAND_START]            		:= (SequencerStatus.CurrentState = E_PackMLState.Starting);
SUPER^.CommandCompletionConditions[INDEX_COMMAND_STOP]             		:= (SequencerStatus.CurrentState = E_PackMLState.Stopping);
SUPER^.CommandCompletionConditions[INDEX_COMMAND_SUSPEND]          		:= (SequencerStatus.CurrentState = E_PackMLState.Suspending);

// Enable/Disable don't have specific PackML states, handle as needed
SUPER^.CommandCompletionConditions[INDEX_COMMAND_ENABLE]           		:= (NOT SUPER^.BaseStatus.Enabled);
SUPER^.CommandCompletionConditions[INDEX_COMMAND_DISABLE]          		:= SUPER^.BaseStatus.Enabled;

_EvaluateCompletionConditions	:= TRUE;
*)
METHOD PROTECTED ABSTRACT _EvaluateCompletionConditions : BOOL
END_METHOD

METHOD PROTECTED _InjectCommandConfiguration : BOOL;
VAR_IN_OUT
	iCommandConfiguration			: ARRAY[*] OF I_CommandConfiguration; // External Dependency			
END_VAR
VAR
    InputLowerBound : DINT;
    InputUpperBound : DINT;
    TargetIndex : DINT;
END_VAR
// External injection still supported for advanced use cases
// Copies configuration data from external source into CommandPermIntlkConfiguration
InputLowerBound := LOWER_BOUND(iCommandConfiguration, 1);
InputUpperBound := UPPER_BOUND(iCommandConfiguration, 1);

// Iterate through target array bounds, mapping to input array
FOR CommandIndexCyclic := LOWER_BOUND(CommandPermIntlkConfiguration,1) TO UPPER_BOUND(CommandPermIntlkConfiguration,1) BY 1 DO
    // Calculate corresponding index in input array
    TargetIndex := CommandIndexCyclic - LOWER_BOUND(CommandPermIntlkConfiguration,1) + InputLowerBound;

    // Check if index is within input array bounds
    IF (TargetIndex >= InputLowerBound) AND (TargetIndex <= InputUpperBound) THEN
        // Validate interface before injection - just check for non-null
        IF (iCommandConfiguration[TargetIndex] <> 0) THEN
            // Copy configuration data from external source
            CommandPermIntlkConfiguration[CommandIndexCyclic].P_CommandConfiguration :=
                iCommandConfiguration[TargetIndex].P_CommandConfiguration;
        ELSE
            // Interface is null
            IF __ISVALIDREF(ComponentConfiguration.BaseConfiguration) THEN
                IF ComponentConfiguration.BaseConfiguration.LogTraceConfiguration.What.xLogToEventLogger THEN
                    TraceWithSeverity(Message := Tc2_Standard.CONCAT('Invalid CommandConfiguration interface at index ', DINT_TO_STRING(TargetIndex)),
                                     Severity := Global.TcEventSeverity.Warning);
                END_IF
            END_IF
        END_IF
        // Note: NULL interfaces are silently ignored (allows partial injection)
    END_IF
END_FOR

ComponentStatus.CommandConfigurationInjected := TRUE;
_InjectCommandConfiguration := TRUE;
END_METHOD

METHOD PROTECTED _InjectPermIntlkConfiguration : BOOL
VAR_IN_OUT
	iPermIntlkConfiguration			: ARRAY[*] OF I_PermIntlkConfiguration; // External Dependency			
END_VAR
VAR
    InputLowerBound : DINT;
    InputUpperBound : DINT;
    TargetIndex : DINT;
END_VAR
// External injection still supported for advanced use cases
// Copies configuration data from external source into CommandPermIntlkConfiguration
InputLowerBound := LOWER_BOUND(iPermIntlkConfiguration, 1);
InputUpperBound := UPPER_BOUND(iPermIntlkConfiguration, 1);

// Iterate through target array bounds, mapping to input array
FOR CommandIndexCyclic := LOWER_BOUND(CommandPermIntlkConfiguration,1) TO UPPER_BOUND(CommandPermIntlkConfiguration,1) BY 1 DO
    // Calculate corresponding index in input array
    TargetIndex := CommandIndexCyclic - LOWER_BOUND(CommandPermIntlkConfiguration,1) + InputLowerBound;

    // Check if index is within input array bounds
    IF (TargetIndex >= InputLowerBound) AND (TargetIndex <= InputUpperBound) THEN
        // Validate interface before injection - just check for non-null
        IF (iPermIntlkConfiguration[TargetIndex] <> 0) THEN
            // Copy configuration data from external source
            CommandPermIntlkConfiguration[CommandIndexCyclic].P_PermIntlkConfiguration :=
                iPermIntlkConfiguration[TargetIndex].P_PermIntlkConfiguration;
        ELSE
            // Interface is null
            IF __ISVALIDREF(ComponentConfiguration.BaseConfiguration) THEN
                IF ComponentConfiguration.BaseConfiguration.LogTraceConfiguration.What.xLogToEventLogger THEN
                    TraceWithSeverity(Message := Tc2_Standard.CONCAT('Invalid PermIntlkConfiguration interface at index ', DINT_TO_STRING(TargetIndex)),
                                     Severity := Global.TcEventSeverity.Warning);
                END_IF
            END_IF
        END_IF
        // Note: NULL interfaces are silently ignored (allows partial injection)
    END_IF
END_FOR

_InjectPermIntlkConfiguration := TRUE;
END_METHOD

METHOD PROTECTED _ObtainAmsNetId
VAR_STAT
	bExecuteEdge : BOOL := FALSE;  // Track execution state for edge triggering
END_VAR
// Validate BaseStatus reference before writing to its fields
IF NOT __ISVALIDREF(ComponentStatus.BaseStatus) THEN
	TraceWithSeverity(Message := 'ComponentStatus.BaseStatus reference is invalid in _ObtainAmsNetId', Severity := Global.TcEventSeverity.Error);
	RETURN;
END_IF

// First call: trigger execution with rising edge
IF NOT bExecuteEdge THEN
	// Clear the memory on first call
	ComponentConfiguration.AmsNetId := '';
	ComponentStatus.AmsNetIdIsValid	:= FALSE;
	bExecuteEdge := TRUE;  // Set to create rising edge
END_IF

GetAmsNetId(
	bExecute:= bExecuteEdge,
	//tTimeOut:= ,
	bBusy=> ComponentStatus.BaseStatus.Busy,
	bError=> ComponentStatus.BaseStatus.Error,
	nErrId=> ComponentStatus.BaseStatus.ErrorID,
	AddrString=> ComponentStatus.AmsNetId
	//AddrBytes=>  ComponentStatus.AmsNetId.AmsNetIdBytes,
);

// Check if function block has completed (not busy and not in first call)
IF NOT GetAmsNetId.bBusy AND bExecuteEdge THEN
	IF NOT GetAmsNetId.bError THEN
		// Validate result
		IF __ISVALIDREF(ComponentStatus.AmsNetId) THEN
			IF (ComponentStatus.AmsNetId <> '') AND (ComponentStatus.AmsNetId <> '0.0.0.0.0.0') THEN
				ComponentStatus.AmsNetIdIsValid	:= TRUE;
				bExecuteEdge := FALSE;  // Reset for next initialization cycle
			END_IF
		ELSE
			TraceWithSeverity(Message := 'AmsNetId Data Reference invalid', Severity := Global.TcEventSeverity.Error);
		END_IF
	ELSE
		// Error occurred - reset edge for potential retry
		bExecuteEdge := FALSE;
	END_IF
END_IF

// Note: ComponentStatus.AmsNetId and ComponentConfiguration.AmsNetId reference the same memory (line 498 in _InitializeReferences)
// The FB writes directly to ComponentConfiguration.AmsNetId through the reference
END_METHOD

METHOD PROTECTED _ProcessCommandQueue
VAR
    oldCmdIndex : DINT;
    oldPriority : DINT;
    newPriority : DINT;
END_VAR
// Guard against multiple queue processing calls per cycle
IF ProcessCommandQueueCalled THEN
	RETURN;
END_IF
ProcessCommandQueueCalled := TRUE;

// Ensure ring buffer exists and has objects
IF (iRingBufferICmd = 0) OR 
   (iRingBufferICmd.P_RingBufferStatus.ObjectCountInBufferPrim = 0) THEN
    RETURN;
END_IF

// Dequeue next command
iRingBufferICmd.RemoveObject();

IF NOT iRingBufferICmd.P_ObjectWasRemoved THEN
    RETURN;
END_IF

// Priority handling - only process if priority is enabled and current command is busy
IF ComponentConfiguration.UseCommandPriority AND ComponentStatus.BaseStatus.Busy THEN
    // Validate removed object before accessing priority
    IF (iRingBufferICmd.P_LastObjectRemoved.iCmdCfg = 0) THEN
        IF __ISVALIDREF(ComponentConfiguration.BaseConfiguration) THEN
            IF ComponentConfiguration.BaseConfiguration.LogTraceConfiguration.What.xLogToEventLogger THEN
                TraceWithSeverity(Message := 'Invalid command configuration in queue', Severity := Global.TcEventSeverity.Warning);
            END_IF
        END_IF
        iRingBufferICmd.ClearStatusFlagRemoved();
        RETURN;
    END_IF

	IF ComponentStatus.iLastCommand <> 0 THEN
		oldCmdIndex := ComponentStatus.iLastCommand.P_CommandStatus.ConfigRef.CommandIndex;
		oldPriority := ComponentStatus.iLastCommand.P_CommandStatus.ConfigRef.Priority;
	END_IF
    newPriority := iRingBufferICmd.P_LastObjectRemoved.iCmdCfg.P_CommandConfiguration.Priority;

    // Debug trace for priority comparison (only if verbose logging enabled)
    IF __ISVALIDREF(ComponentConfiguration.BaseConfiguration) THEN
        IF ComponentConfiguration.BaseConfiguration.LogTraceConfiguration.What.xLogToEventLogger THEN
            TraceWithSeverity(Message := Tc2_Standard.CONCAT('Priority check: old=',
                             Tc2_Standard.CONCAT(DINT_TO_STRING(oldPriority),
                             Tc2_Standard.CONCAT(' new=', DINT_TO_STRING(newPriority)))),
                             Severity := Global.TcEventSeverity.Verbose);
        END_IF
    END_IF
    
    // Check if a command is currently running with valid interfaces
    IF (oldCmdIndex >= LOWER_BOUND(iCommands, 1)) AND
       (oldCmdIndex <= UPPER_BOUND(iCommands, 1)) AND
       (iCommands[oldCmdIndex] <> 0) THEN
        
        IF newPriority < oldPriority THEN
            // Lower priority should wait → re-enqueue
            iRingBufferICmd.AddObject(RefObject := iRingBufferICmd.P_LastObjectRemoved);

            // Check if re-enqueue succeeded
            IF NOT iRingBufferICmd.P_ObjectWasAdded THEN
                IF __ISVALIDREF(ComponentConfiguration.BaseConfiguration) THEN
                    IF ComponentConfiguration.BaseConfiguration.LogTraceConfiguration.What.xLogToEventLogger THEN
                        TraceWithSeverity(Message := 'Failed to re-enqueue lower priority command - buffer may be full', Severity := Global.TcEventSeverity.Error);
                    END_IF
                END_IF
            ELSE
                // Successfully re-added - clear the flag
                iRingBufferICmd.ClearStatusFlagAdded();
            END_IF

            iRingBufferICmd.ClearStatusFlagRemoved();
            RETURN;
        ELSIF newPriority > oldPriority THEN
            // Higher priority preempts - abort current command
            iCommands[oldCmdIndex].Abort();
            IF __ISVALIDREF(ComponentConfiguration.BaseConfiguration) THEN
                IF ComponentConfiguration.BaseConfiguration.LogTraceConfiguration.What.xLogToEventLogger THEN
                    TraceWithSeverity(Message := Tc2_Standard.CONCAT('Preempting command[',
                                     Tc2_Standard.CONCAT(DINT_TO_STRING(oldCmdIndex), '] with higher-priority request')),
                                     Severity := Global.TcEventSeverity.Info);
                END_IF
            END_IF
        END_IF
        // If priorities are equal (newPriority = oldPriority), current command continues without abort
    END_IF
ELSE
    // Debug: Log when priority checking is skipped (only if verbose logging enabled)
    IF __ISVALIDREF(ComponentConfiguration.BaseConfiguration) THEN
        IF ComponentConfiguration.BaseConfiguration.LogTraceConfiguration.What.xLogToEventLogger THEN
            IF NOT ComponentConfiguration.UseCommandPriority THEN
                TraceWithSeverity(Message := 'Priority check skipped: UseCommandPriority=FALSE', Severity := Global.TcEventSeverity.Verbose);
            ELSIF NOT ComponentStatus.BaseStatus.Busy THEN
                TraceWithSeverity(Message := 'Priority check skipped: Component not busy', Severity := Global.TcEventSeverity.Verbose);
            END_IF
        END_IF
    END_IF
END_IF

// Validate command before execution
IF (iRingBufferICmd.P_LastObjectRemoved.iCmd = 0) THEN
    IF __ISVALIDREF(ComponentConfiguration.BaseConfiguration) THEN
        IF ComponentConfiguration.BaseConfiguration.LogTraceConfiguration.What.xLogToEventLogger THEN
            TraceWithSeverity(Message := 'Invalid command interface in dequeued object', Severity := Global.TcEventSeverity.Error);
        END_IF
    END_IF
    iRingBufferICmd.ClearStatusFlagRemoved();
    RETURN;
END_IF

// Set status to Accepted and trigger execution (Execute() no longer sets redundant status)
IF iRingBufferICmd.P_LastObjectRemoved.iCmd <> 0 AND iRingBufferICmd.P_LastObjectRemoved.iCmdCfg <> 0 THEN
	iRingBufferICmd.P_LastObjectRemoved.iCmd.Execute();
	ComponentStatus.iLastCommand			 	:= iRingBufferICmd.P_LastObjectRemoved.iCmd;
	ComponentStatus.iLastCommandConfiguration	:= iRingBufferICmd.P_LastObjectRemoved.iCmdCfg;

	// Command monitoring is handled by _MonitorCommandCompletion() in the cyclic logic
END_IF

// Clear removal flag
iRingBufferICmd.ClearStatusFlagRemoved();
END_METHOD

METHOD PROTECTED _TryRehashDispatchIndex : BOOL
VAR_INPUT
    sCommandPOUName : STRING;
END_VAR
// IF _ZaberAxisConfigurationFW744 = 0 THEN
//     TraceWithSeverity('Hash table is NULL – command aborted', Severity := Global.TcEventSeverity.Error);
//     _TryRehashDispatchIndex := FALSE;
//     RETURN;
// END_IF

//Rehash
ComponentStatus.MethodDispatch := GetIndexByPOUName(NameIn := sCommandPOUName);

IF NOT ((ComponentStatus.MethodDispatch >= LOWER_BOUND(Commands, 1)) AND
        (ComponentStatus.MethodDispatch <= UPPER_BOUND(Commands, 1))) THEN
    	IF __ISVALIDREF(ComponentConfiguration.BaseConfiguration) THEN
    		IF ComponentConfiguration.BaseConfiguration.LogTraceConfiguration.What.xLogToEventLogger THEN
    			TraceWithSeverity('Hashing failed.  Interface valid but hash table may have no initial insert', Severity := Global.TcEventSeverity.Error);
    		END_IF
    	END_IF

    _TryRehashDispatchIndex := FALSE;
    RETURN;
END_IF

_TryRehashDispatchIndex := TRUE;
END_METHOD

METHOD PROTECTED _UpdateBusyStatus
// Derive overall Busy flag after command completion
// This ensures Busy status accurately reflects commands that completed in this cycle

// Validate reference before accessing
IF NOT __ISVALIDREF(ComponentStatus.BaseStatus) THEN
	RETURN;
END_IF

ComponentStatus.BaseStatus.Busy := FALSE;
FOR CommandIndexExit := LOWER_BOUND(Commands, 1) TO UPPER_BOUND(Commands, 1) DO
    IF iCommands[CommandIndexExit] <> 0 THEN
	IF iCommands[CommandIndexExit].Busy THEN
		ComponentStatus.BaseStatus.Busy := TRUE;
		EXIT;				// any busy
	ELSE
		ComponentStatus.BaseStatus.Busy	:= FALSE;
	END_IF
    END_IF
END_FOR
END_METHOD

(* Example implementation from FB_Actuator:
IF ActuatorStatus.ExtendOutput AND NOT ActuatorStatus.RetractOutput THEN
	ActuatorStatus.ActuatorState	:= E_ActuatorState.Extended;
ELSIF ActuatorStatus.RetractOutput AND NOT ActuatorStatus.ExtendOutput THEN
	ActuatorStatus.ActuatorState	:= E_ActuatorState.Retracted;
ELSE
	ActuatorStatus.ActuatorState	:= E_ActuatorState.Indeterminate;
END_IF

_UpdateComponentStatus := THIS^;*)

METHOD PROTECTED ABSTRACT _UpdateComponentStatus : I_ComponentFull
END_METHOD

METHOD CyclicLogic
SUPER^.CyclicLogic();

